FUNCTION_BLOCK "GCS7_E_MDDx_DP"	// FB 37
TITLE = MDDx Profibus Communication
//  
//COPYRIGHT:    (C) 1998  BUHLER AG, CH-9240 UZWIL, SWITZERLAND
//
//PRODUCT:      GCS7R1
//
//TITLE:        Element Control MDDx Profibus Communication
//
//REVISION:     11
//
//-------------------------------------------------------------------------
//
//IDENT:        AUTHOR:             DEPT:                      DATE:
//
//FB37.3.3      A. Egli             BASE                       30-Mar-2009
//              -PCD: OType=1037
//FB37.3.3      A. Egli             BASE                       16-Dec-2008
//              -Gap adjustement MDDR/T (GCS7R2 3.3)
//FB37.2.1      A. Egli             BASE                       25-Mar-2008
//              Len UDT SSW_MDDX_DP_Alarm is 6 Byte
//FB37.2.0      A. Egli             CT3                        25-Feb-2008
//              - New tagname for digital inputs Status.InpDI_0x
//              - Delete Status if OutComFault
//FB37.1.2      A. Egli             CT3                        21-Nov-2007
//              Message 42=A072CANDOUT
//FB37.1.1      A. Egli             CT3                        19-Nov-2006
//              Copy also AlarmNo > 74
//FB37.1.0      A. Egli             CT3                        11-Jun-2005
//              New Release R1
//
//-------------------------------------------------------------------------
//
//PURPOSE:      MANUAL : see [SSW-EL-MDDX_MAN_en]
//
//RESTRICTIONS: S7
//              ParFault and ParWarning may be set together!
//
//
//-------------------------------------------------------------------------
//=======================================================
//Log Message: 
//------------------------------------------------------
//
//=======================================================
//StCode:  State Communication               
//------------------------------------------------------
//43  StComFault.Local
// 3  StComOk                    
//32  StFault                 
//=======================================================
//StCode:  State Passage
//------------------------------------------------------
// 1  StDisengaged 
//11  StDisengaged.Warning 
//41  StDisengaged.DPFault
// 4  StEngaged
//14  StEngaged.Warning 
//44  StEngaged.DPFault
//32  StFault                 
//
//
AUTHOR : EA
FAMILY : GCS7LL
NAME : MDDxDP
VERSION : 3.4
VAR
  StCode : INT ;	//Element state code
  spare20 : BOOL ;
  spare21 : BOOL ;
  InOverrideHL : BOOL ;	//Override HL Inlet
  CmdNewJob : BOOL ;	//Send Target Value to LC, even if in manual mode
  CmdNewValue : BOOL ;	//Send Target Values
  spare25 : BOOL ;
  spare26 : BOOL ;
  spare27 : BOOL ;
  spare30 : BOOL ;
  spare31 : BOOL ;
  spare32 : BOOL ;
  CmdFaultReset : BOOL ;	//Command to reset fault
  InLocal : BOOL ;	//1= Local mode (no fault by start with service switch)
  spare35 : BOOL ;	//Warning is active
  spare36 : BOOL ;
  spare37 : BOOL ;
  InSimulation : BOOL ;	//Simulation with DPSim
  OutComFault : BOOL ;	//Communication fault
  VarEdgeStFault : BOOL ;
  OutWarning : BOOL ;
  OutFaultRelevant : BOOL ;	//Relavant faultfor group
  OutEdgeComFault : BOOL ;	//Alarm reason
  spare46 : BOOL ;
  spare47 : BOOL ;
  spare50 : BOOL ;
  spare51 : BOOL ;
  StOk : BOOL ;	//Element is ok
  spare53 : BOOL ;
  StFault : BOOL ;	//Element has a communication or device fault
  PCWrite : STRUCT
   Hsk : STRUCT
    AckRegisterSide1 : BOOL ;	//Acknowledge save recipe
    AckRollChangeDoneSide1 : BOOL ;	//Acknowledge roll change
    AckRegisterSide2 : BOOL ;	//Acknowledge save recipe
    AckRollChangeDoneSide2 : BOOL ;	//Acknowledge roll change
    Ack600CalibrationSide1 : BOOL ;	//Acknowledge 600 calibration
    Ack600CalibrationSide2 : BOOL ;	//Acknowledge 600 calibration
   END_STRUCT ;
  END_STRUCT ;
  PCRead : STRUCT
   Hsk : STRUCT
    ReqRegisterSide1 : BOOL ;	//Announcement save recipe
    ReqRollChangeDoneSide1 : BOOL ;	//Announcement roll change has be done
    ReqRegisterSide2 : BOOL ;	//Announcement save recipe
    ReqRollChangeDoneSide2 : BOOL ;	//Announcement roll change has be done
    Req600CalibrationSide1 : BOOL ;	//Announcement 600 calibration
    Req600CalibrationSide2 : BOOL ;	//Announcement 600 calibration
   END_STRUCT ;
  END_STRUCT ;
  Side1 : STRUCT
   StCode : INT ;
   InEnableDosing : BOOL ;	//Signal to engage the rolls and start dosing
   InRestdischarge : BOOL ;	//Signal to activate restdischarge mode
   CmdNewJob : BOOL ;	//Send Target Value to LC, even if in manual mode
   CmdNewValue : BOOL ;	//Send new Values to LC
   OutLCFault : BOOL ;	//LC has a relevant fault
   OutLCWarning : BOOL ;	//LC has a relevant fault
   OutAlarmNoValid : BOOL ;
   OutManual : BOOL ;	//LC Manual Mode
   VarEdgeStFault : BOOL ;
   StDisenaged : BOOL ;	//Element is ok
   StEngaged : BOOL ;	//Element is ok
   StFault : BOOL ;	//Element has a communication or device fault
   In : STRUCT 	//Only without MDEF
    InRollsUpCurrent : INT ;	//de: Aktuelle Stromaufnahme Motor 1 [0.1 A]
    InRollsLowCurrent : INT ;	//de: Aktuelle Stromaufnahme Motor 2 [0.1 A]
    InGapTopLeft : INT ;	//de:  Sollwert Mahlspalt oben links
    InGapTopRight : INT ;	//de:  Sollwert Mahlspalt oben rechts
    InGapBottomLeft : INT ;	//de:  Sollwert Mahlspalt unten links
    InGapBottomRight : INT ;	//de:  Sollwert Mahlspalt unten rechts
    InRollsLowUsed : BOOL ;	//MDDT: 1=Engage also lower rolls
    InRollsUpUsed : BOOL ;	//MDDT: 1=Engage also upper rolls
    InGapAdjustment : INT ;	//10=OFF,11=AUT,12=MAN,13=LOC,14=RCHG,0=nothing
   END_STRUCT ;
   Out : STRUCT 	//Only without MDEF
    OutRollsUpLoad : INT ;	//Is read from LC [%]
    OutRollsUpCurrent : INT ;	//Is read from LC [0.1 A]
    OutRollsLowLoad : INT ;	//Is read from LC [%]
    OutRollsLowCurrent : INT ;	//Is read from LC [0.1 A]
    OutFeedRollSpeed : INT ;	//Is read from LC [Hz]
    OutGrindingRollsUpSpeed : INT ;	//Is read from LC [0..999 RPM]
    OutGrindingRollsLowSpeed : INT ;	//Is read from LC [0..999 RPM]
    spare : INT ;
    OutAlarmNo : INT ;	//Is read from LC [0..9999]
    OutGapAdjustmentStatus : INT ;	//10=OFF,11=AUT,12=MAN,13=LOC,14=RCHG
    OutGapTopLeftAct : INT ;	//de:  Istwert Mahlspalt oben links
    OutGapTopRightAct : INT ;	//de:  Istwert Mahlspalt oben rechts
    OutGapBottomLeftAct : INT ;	//de:  Istwert Mahlspalt unten links
    OutGapBottomRightAct : INT ;	//de:  Istwert Mahlspalt unten rechts
    OutProductLevel : INT ;	//Is read from LC [+-500]
    OutTemperatureHoot : INT ;	//Is read from LC [°C]
    OutRunningTimeEngage : INT ;	//Is read from LC [h]
    OutRunningTimeRollsUp : INT ;	//Is read from LC [h]
    OutRunningTimeRollsLow : INT ;	//Is read from LC [h]
    OutCntEngage : INT ;	//Is read from LC []
    OutStatus : STRUCT 	//Is read from LC
     OutMDDR : BOOL ;
     OutHLBackupLeft : BOOL ;
     OutHLBackupRight : BOOL ;
    END_STRUCT ;
    OutLCAlarm : UDT 20373;
    tmpLCAlarm : UDT 20373;
   END_STRUCT ;
   OutTimeFaulted : DINT ;	//[s] Not errasable time "Faulted"
   OutCntFault : DINT ;	//Not errasable counter of faults
  END_STRUCT ;
  Side2 : STRUCT
   StCode : INT ;
   InEnableDosing : BOOL ;	//Signal to engage the rolls and start dosing
   InRestdischarge : BOOL ;	//Signal to activate restdischarge mode
   CmdNewJob : BOOL ;	//Send Target Value to LC, even if in manual mode
   CmdNewValue : BOOL ;	//Send new Values to LC
   OutLCFault : BOOL ;	//LC has a relevant fault
   OutLCWarning : BOOL ;	//LC has a relevant fault
   OutAlarmNoValid : BOOL ;
   OutManual : BOOL ;	//LC Manual Mode
   VarEdgeStFault : BOOL ;
   StDisenaged : BOOL ;	//Element is ok
   StEngaged : BOOL ;	//Element is ok
   StFault : BOOL ;	//Element has a communication or device fault
   In : STRUCT 	//Only without MDEF
    InRollsUpCurrent : INT ;	//de: Aktuelle Stromaufnahme Motor 1 [0.1 A]
    InRollsLowCurrent : INT ;	//de: Aktuelle Stromaufnahme Motor 2 [0.1 A]
    InGapTopLeft : INT ;	//de:  Sollwert Mahlspalt oben links
    InGapTopRight : INT ;	//de:  Sollwert Mahlspalt oben rechts
    InGapBottomLeft : INT ;	//de:  Sollwert Mahlspalt unten links
    InGapBottomRight : INT ;	//de:  Sollwert Mahlspalt unten rechts
    InRollsLowUsed : BOOL ;	//MDDT: 1=Engage also lower rolls
    InRollsUpUsed : BOOL ;	//MDDT: 1=Engage also upper rolls
    InGapAdjustment : INT ;	//10=OFF,11=AUT,12=MAN,13=LOC,14=RCHG,0=nothing
   END_STRUCT ;
   Out : STRUCT 	//Only without MDEF
    OutRollsUpLoad : INT ;	//Is read from LC [%]
    OutRollsUpCurrent : INT ;	//Is read from LC [0.1 A]
    OutRollsLowLoad : INT ;	//Is read from LC [%]
    OutRollsLowCurrent : INT ;	//Is read from LC [0.1 A]
    OutFeedRollSpeed : INT ;	//Is read from LC [HZ]
    OutGrindingRollsUpSpeed : INT ;	//Is read from LC [0..999 RPM]
    OutGrindingRollsLowSpeed : INT ;	//Is read from LC [0..999 RPM]
    spare : INT ;
    OutAlarmNo : INT ;	//Is read from LC [0..9999]
    OutGapAdjustmentStatus : INT ;	//0=Off;1=Manual;2=Automatic;3=Referencing;4=Aligment;5=Save
    OutGapTopLeftAct : INT ;	//de:  Istwert Mahlspalt oben links
    OutGapTopRightAct : INT ;	//de:  Istwert Mahlspalt oben rechts
    OutGapBottomLeftAct : INT ;	//de:  Istwert Mahlspalt unten links
    OutGapBottomRightAct : INT ;	//de:  Istwert Mahlspalt unten rechts
    OutProductLevel : INT ;	//Is read from LC [+-500]
    OutTemperatureHoot : INT ;	//Is read from LC [°C]
    OutRunningTimeEngage : INT ;	//Is read from LC [h]
    OutRunningTimeRollsUp : INT ;	//Is read from LC [h]
    OutRunningTimeRollsLow : INT ;	//Is read from LC [h]
    OutCntEngage : INT ;	//Is read from LC []
    OutStatus : STRUCT 	//Is read from LC
     OutMDDR : BOOL ;
     OutHLBackupLeft : BOOL ;
     OutHLBackupRight : BOOL ;
    END_STRUCT ;
    OutLCAlarm : UDT 20373;
    tmpLCAlarm : UDT 20373;
   END_STRUCT ;
   OutTimeFaulted : DINT ;	//[s] Not errasable time "Faulted"
   OutCntFault : DINT ;	//Not errasable counter of faults
  END_STRUCT ;
  Side1Divide : STRUCT
   StCode : INT ;
   OutLCFault : BOOL ;	//LC has a relevant fault
   OutLCWarning : BOOL ;	//LC has a relevant fault
   OutAlarmNoValid : BOOL ;
   VarEdgeStFault : BOOL ;
   StDisenaged : BOOL ;	//Element is ok
   StEngaged : BOOL ;	//Element is ok
   StFault : BOOL ;	//Element has a communication or device fault
   Out : STRUCT
    OutProductLevel : INT ;	//Is read from LC [+-500]
    OutFeedRollSpeed : INT ;	//Is read from LC [0..999 RPM]
    OutHLInlet : BOOL ;	//de:Einlaufsonde Left
    OutAlarmNo : INT ;	//Is read from LC [0..9999]
    OutLCAlarm : UDT 20373;
    tmpLCAlarm : UDT 20373;
   END_STRUCT ;
   OutTimeFaulted : DINT ;	//[s] Not errasable time "Faulted"
   OutCntFault : DINT ;	//Not errasable counter of faults
  END_STRUCT ;
  Side2Divide : STRUCT
   StCode : INT ;
   OutLCFault : BOOL ;	//LC has a relevant fault
   OutLCWarning : BOOL ;	//LC has a relevant fault
   OutAlarmNoValid : BOOL ;
   VarEdgeStFault : BOOL ;
   StDisenaged : BOOL ;	//Element is ok
   StEngaged : BOOL ;	//Element is ok
   StFault : BOOL ;	//Element has a communication or device fault
   Out : STRUCT
    OutProductLevel : INT ;	//Is read from LC [+-500]
    OutFeedRollSpeed : INT ;	//Is read from LC [0..999 RPM]
    OutHLInlet : BOOL ;	//de:Einlaufsonde Left
    OutAlarmNo : INT ;	//Is read from LC [0..9999]
    OutLCAlarm : UDT 20373;
    tmpLCAlarm : UDT 20373;
   END_STRUCT ;
   OutTimeFaulted : DINT ;	//[s] Not errasable time "Faulted"
   OutCntFault : DINT ;	//Not errasable counter of faults
  END_STRUCT ;
  OutAlarmNoLog : INT ;	//Last textnumber send to log
  OutTimeFaulted : DINT ;	//[s] Not errasable time "Faulted"
  OutCntFault : DINT ;	//Not errasable counter of faults
  Command : STRUCT
   S1Start : BOOL ;	//de: Start/Stop Links
   spare01 : BOOL ;
   S1RestDischarge : BOOL ;	//de: Restentleeren Links
   spare03 : BOOL ;
   spare04 : BOOL ;
   S1AckNewGapStatus : BOOL ;	//Acknowledge reading data
   spare06 : BOOL ;
   AcceptNewDataReady : BOOL ;	//de: Quittierung neue Werte Bereit
   S2Start : BOOL ;	//de: Start/Stop Rechts
   spare11 : BOOL ;
   S2RestDischarge : BOOL ;	//de: Restentleeren Rechts
   spare13 : BOOL ;
   spare14 : BOOL ;
   S2AckNewGapStatus : BOOL ;	//Acknowledge reading data
   spare16 : BOOL ;
   spare17 : BOOL ;	//de: Quittierung neue Werte Bereit
   spare20 : BYTE ;
   CommandReady : BOOL ;	//de: Steuersignale gültig
   spare31 : BOOL ;
   spare32 : BOOL ;
   spare33 : BOOL ;
   spare34 : BOOL ;
   ResetAlarm : BOOL ;	//de: Alarm löschen
   NewSendData : BOOL ;	//de: Aenderung Sendedaten
   AcceptNewRcvData : BOOL ;	//de: Quittierung Aenderung Empfangsdatensatz
  END_STRUCT ;
  Status : STRUCT
   S1Operation : BOOL ;	//de: Betrieb
   S1Disengaged : BOOL ;	//de: 1=Ausgerückt
   S1RestdischargeLocal : BOOL ;	//de: 1=Restentleeren Local
   S1DisengagedManual : BOOL ;	//Rolls manually disengaged: 1=Manually disengaged
   S1EnableMotors : BOOL ;	//de: Freigabe Mahlmotoren
   spare05 : BOOL ;
   spare06 : BOOL ;
   NewDataReady : BOOL ;	//de: Neue Werte Bereit
   S2Operation : BOOL ;	//de: Betrieb
   S2Disengaged : BOOL ;	//de: 1=Ausgerückt
   S2RestdischargeLocal : BOOL ;	//de: 1=Restentleeren Local
   S2DisengagedManual : BOOL ;	//Rolls manually disengaged: 1=Manually disengaged
   S2EnableMotors : BOOL ;	//de: Freigabe Mahlmotoren
   spare15 : BOOL ;
   spare16 : BOOL ;
   spare17 : BOOL ;	//de: Neue Werte Bereit
   InpDI_0_4 : BOOL ;	//DI 0.4: Default: Side 1 HL Inlet
   InpDI_0_5 : BOOL ;	//DI 0.5: Default: Side 1 HL Outlet 1
   InpDI_0_6 : BOOL ;	//DI 0.6: Default: Side 1 HL Outlet 2
   InpDI_0_7 : BOOL ;	//DI 0.7: Default: Side 1 HL Outlet 3
   InpDI_0_16 : BOOL ;	//DI 0.16: Default: Side 2 HL Inlet
   InpDI_0_17 : BOOL ;	//DI 0.17: Default: Side 2 HL Outlet 1
   InpDI_0_18 : BOOL ;	//DI 0.18: Default: Side 2 HL Outlet 2
   InpDI_0_19 : BOOL ;	//DI 0.19: Default: Side 2 HL Outlet 3
   InpDI_0_0 : BOOL ;	//DI0.0 Terminal X5:2
   InpDI_0_1 : BOOL ;	//DI0.1 Terminal X5:3
   InpDI_0_2 : BOOL ;	//DI0.2 Terminal X5:4
   RemoteControl : BOOL ;	//de: Sollwertvorgabe Remote
   WrongValue : BOOL ;	//de: Falscher Sollwert
   SumFault : BOOL ;	//de: Sammelalarm
   AcceptNewSendData : BOOL ;	//de: Quittierung Aenderung Sendedaten
   NewRcvData : BOOL ;	//de: Aenderung Empfangsdaten
  END_STRUCT ;
  Par : STRUCT
   ParObjectNo : INT ;	//Is used for communication with PC, e.g. for message
   ParMsgType : INT ;	//Is used for message (translation of state)
   ParHornCode : INT ;	//Is used by horn module
   ParLogOff : BOOL ;	//Report is off
   ParSide1Divided : BOOL ;	//Side 1 is divided
   ParSide2Divided : BOOL ;	//Side 2 is divided
   ParFilter : UDT 20373;	//Filter to alarm 1=Ignore alarm
   ParFilterWarning : UDT 20373;	//Filter to set alarm type (0=Fault;Suspend/1=Warning)
   ParIOByteNo : INT ;	//PROFIBUS: Address of first input and output byte
   HelpFlags : STRUCT
    CmdNewValueS1 : BOOL ;
    CmdNewValueS2 : BOOL ;
    CmdFaultReset : BOOL ;
    OutTestNewAlarm : BOOL ;	//Aux. signal to retry fault message
    OutComFaultRead : BOOL ;
    OutComFaultSend : BOOL ;
   END_STRUCT ;
   OutNoSndDataSet : BYTE ;	//de: Nummer Sendedatensatz
   OutIdxSndDataSet : BYTE ;	//de: Index Sendedatensatz
   OutNoRcvDataSet : BYTE ;	//de: Nummer Sendedatensatz
   OutIdxRcvDataSet : BYTE ;	//de: Index Sendedatensatz
   spare1 : DINT ;
  END_STRUCT ;
END_VAR
VAR_TEMP
  tmpAddrOffset : DWORD ;	//store the Instance Pointer
  tmpLOGvalue : WORD ;	//LOG value
  tmpCommand : INT ;
  tmpFault : BOOL ;
  tmpWarning : BOOL ;
  tmpLocal : BOOL ;
  tmpHornOn : BOOL ;
  tmpSendDone : BOOL ;	//Send Index is Equal receive Index
  tmpBit : BOOL ;
  tmpPxFault : BOOL ;
  tmpPxWarning : BOOL ;
  tmpPxAlarmNoValid : BOOL ;
  tmpAllAlarmNoValide : BOOL ;
  tmpAddrParFilter : DWORD ;	//Pointer to ParFilter
  tmpAddrParFilterWarning : DWORD ;	//Pointer to ParFilterWarning
  tmpIdx : INT ;
  tmpNewAlarm : UDT 20373;
  tmpOldAlarm : UDT 20373;
  tmpParFilterWarning : UDT 20373;
  tmpInt : INT ;
  tmpAddr : WORD ;
  tmpAddrIO : DINT ;
  tmpReturn : INT ;
  DPData : STRUCT
   StatusCommand : DWORD ;
   NoSndDataSet : BYTE ;	//de: Nummer Sendedatensatz
   IdxSndDataSet : BYTE ;	//de: Index Sendedatensatz
   NoRcvDataSet : BYTE ;	//de: Nummer Empfangsdatensatz
   IdxRcvDataSet : BYTE ;	//de: Index Empfangsdatensatz
   Data : STRUCT
    Byte8_9 : INT ;
    Byte10_11 : INT ;
    Byte12_13 : INT ;
    Byte14_15 : INT ;
    Byte16_17 : INT ;
    Byte18_19 : INT ;
    Byte20_21 : INT ;
    Byte22 : BYTE ;
    Byte23 : BYTE ;
   END_STRUCT ;
  END_STRUCT ;
  DPData16 : STRUCT
   StatusCommand : DWORD ;
   NoSndDataSet : BYTE ;	//de: Nummer Sendedatensatz
   IdxSndDataSet : BYTE ;	//de: Index Sendedatensatz
   NoRcvDataSet : BYTE ;	//de: Nummer Empfangsdatensatz
   IdxRcvDataSet : BYTE ;	//de: Index Empfangsdatensatz
   Data : ARRAY  [1 .. 4 ] OF DINT ;
  END_STRUCT ;
  DPData_Alarm120 : ARRAY  [0 .. 127 ] OF BOOL ;
  DPData_Alarm121 : ARRAY  [127 .. 255 ] OF BOOL ;
  tmpAddrOut_OutLCAlarm : DWORD ;
  tmpAddrOut_tmpLCAlarm : DWORD ;
END_VAR
BEGIN
NETWORK
TITLE =  Start Global
      TAR2;
      L     DW#16#FFFFFF;
      AD;
      T     #tmpAddrOffset;	//-->Addr Para
      L     P##Par;	//[3.1]
      +D;	//[3.1]
      L     P#8.0;
      +D;
      T     #tmpAddrParFilter;	//-->Pointer to Par.ParFilter
      L     P#6.0;
      +D;
      T     #tmpAddrParFilterWarning;	//-->Pointer to Par.ParFilterWarning
      SET;
      R     #tmpHornOn;
NETWORK
TITLE = PC Control
//=== Test Object number =====================
      L     "SYS_DirectCtrlDB".PC.ObjectNo;	//PCControl.ObjectNo
      L     #Par.ParObjectNo;	//Input ObjectNo
      <>I;
      JC    Ctrl;
//=== Test OType      ========================
      L     1037;	//Input object type
      L     "SYS_DirectCtrlDB".PC.ObjectType;	//PCControl.ObjectType
      <>I;
      JC    Ctrl;
//=== Test Handshake =========================
      A     "SYS_DirectCtrlDB".PC.Hsk.FExamine;	// Handshake.FExamine
      JC    pExa;
      A     "SYS_DirectCtrlDB".PC.Hsk.FDefineCmd;	// Handshake.FDefineCmd
      JC    pCmd;
      A     "SYS_DirectCtrlDB".PC.Hsk.FDefinePara;	// Handshake.FDefinePara
      JC    pPar;
      JU    pIni;
pIni: L     2;	//FcInit
      UC    "SYS_DirectCtrl";
      JU    Ctrl;
//Write parameter 
pPar: NOP   0;
//Write new commands from PC to Interface of group 
pCmd: A     "SYS_DirectCtrlDB".PC.Cmd1[11];	//CmdFaultReset
      S     #CmdFaultReset;
//------------------------------------------
pExa: NOP   0;
      TAR2;	// Address Dynamic datas
      T     "SYS_DirectCtrlDB".GC.InDynAddr;	// -->PCControl.GC.InDynAddr
      L     288;	// Length Dynamic datas
      T     "SYS_DirectCtrlDB".GC.InDynLen;	// -->PCControl.GC.InDynLen
      L     0;
      T     "SYS_DirectCtrlDB".GC.InParaAddr;	// -->PCControl.GC.InParaAddr
      T     "SYS_DirectCtrlDB".GC.InParaLen;	// -->PCControl.GC.InParaLen
      L     1;	// Code FcExamine
      UC    "SYS_DirectCtrl";
      L     11;	//Revision
      T     "SYS_DirectCtrlDB".GC.Revision;
Ctrl: NOP   0;
NETWORK
TITLE = (Profibus) Read data and store Data 
      L     #Par.ParIOByteNo;
      T     #tmpAddr;
      A     #InSimulation;
      JC    rSim;
      CALL  "SIEMENS_DPRD_DAT" (
           LADDR                    := #tmpAddr,
           RET_VAL                  := #tmpReturn,
           RECORD                   := #DPData);
      L     #tmpReturn;
      L     0;
      <>I;
      =     #Par.HelpFlags.OutComFaultRead;
      JC    rcv0;
      JU    rDP;
//read from Simulation
rSim: R     #Par.HelpFlags.OutComFaultRead;
      A     "GCS7_Gr_SimDPtoImage";
      L     P#I 0.0;
      JC    rDB1;
      OPN   "TEST_IOSimuliInput";
      L     P#DBX 0.0;
rDB1: L     #Par.ParIOByteNo;
      SLD   3;
      +D;
      T     #tmpAddrIO;
      LAR1  #tmpAddrIO;
      L     D [AR1,P#0.0];
      T     #DPData.StatusCommand;
      LAR1  #tmpAddrIO;
      L     D [AR1,P#4.0];
      LAR1  P##DPData;
      T     LD [AR1,P#4.0];
      LAR1  #tmpAddrIO;
      L     D [AR1,P#8.0];
      LAR1  P##DPData;
      T     LD [AR1,P#8.0];
      LAR1  #tmpAddrIO;
      L     D [AR1,P#12.0];
      LAR1  P##DPData;
      T     LD [AR1,P#12.0];
      LAR1  #tmpAddrIO;
      L     D [AR1,P#16.0];
      LAR1  P##DPData;
      T     D [AR1,P#16.0];
      LAR1  #tmpAddrIO;
      L     D [AR1,P#20.0];
      LAR1  P##DPData;
      T     D [AR1,P#20.0];
//===Test Send Data
rDP:  L     #DPData.NoSndDataSet;
      L     #Par.OutNoSndDataSet;
      ==I;
      A(;
      L     #DPData.IdxSndDataSet;
      L     #Par.OutIdxSndDataSet;
      ==I;
      );
      =     #tmpSendDone;
//==Copy Status===============
      L     #DPData.NoRcvDataSet;
      L     0;
      ==I;
      JC    R01A;
      CALL  "SIEMENS_BLKMOV" (
           SRCBLK                   := #DPData.StatusCommand,
           RET_VAL                  := #tmpReturn,
           DSTBLK                   := #Status);
      AN    #Status.NewRcvData;
      A     #InSimulation;
      JC    rcv0;
//===============================
//Answer Dataset 001
      L     #DPData.NoRcvDataSet;
      L     1;
      <>I;
      JC    r02;
//Answer Dataset 001 Index 1
      L     #DPData.IdxRcvDataSet;
      L     1;
      <>I;
      JC    r01B;
      L     #DPData.Data.Byte8_9;
      T     #Side1.Out.OutRollsUpLoad;
      L     #DPData.Data.Byte10_11;
      T     #Side1.Out.OutRollsUpCurrent;
      L     #DPData.Data.Byte12_13;
      T     #Side1.Out.OutRollsLowLoad;
      L     #DPData.Data.Byte14_15;
      T     #Side1.Out.OutRollsLowCurrent;
      L     #DPData.Data.Byte16_17;
      T     #Side1.Out.OutFeedRollSpeed;
      L     #DPData.Data.Byte18_19;
      T     #Side1.Out.OutGrindingRollsUpSpeed;
      L     #DPData.Data.Byte20_21;
      T     #Side1.Out.OutGrindingRollsLowSpeed;
      L     #DPData.Data.Byte23;
      T     #Side1.Out.OutAlarmNo;
      JU    R01B;
//Answer Dataset 001 Index 2
r01B: L     #DPData.IdxRcvDataSet;
      L     2;
      <>I;
      JC    r01C;
      L     #DPData.Data.Byte8_9;
      T     #Side2.Out.OutRollsUpLoad;
      L     #DPData.Data.Byte10_11;
      T     #Side2.Out.OutRollsUpCurrent;
      L     #DPData.Data.Byte12_13;
      T     #Side2.Out.OutRollsLowLoad;
      L     #DPData.Data.Byte14_15;
      T     #Side2.Out.OutRollsLowCurrent;
      L     #DPData.Data.Byte16_17;
      T     #Side2.Out.OutFeedRollSpeed;
      L     #DPData.Data.Byte18_19;
      T     #Side2.Out.OutGrindingRollsUpSpeed;
      L     #DPData.Data.Byte20_21;
      T     #Side2.Out.OutGrindingRollsLowSpeed;
      L     #DPData.Data.Byte23;
      T     #Side2.Out.OutAlarmNo;
      JU    R01C;
//Answer Dataset 001 Index 3
r01C: L     #DPData.IdxRcvDataSet;
      L     3;
      <>I;
      JC    r02;
//--Side1 Ext
      L     #DPData.Data.Byte8_9;
      T     #Side1Divide.Out.OutProductLevel;
      L     #DPData.Data.Byte10_11;
      T     #Side1Divide.Out.OutFeedRollSpeed;
      L     #DPData.Data.Byte12_13;
      T     #Side1Divide.Out.OutAlarmNo;
      L     #DPData.Data.Byte23;
      L     2#1;
      AW;
      L     0;
      <>I;
      =     #Side1Divide.Out.OutHLInlet;
//--Side2 Ext
      L     #DPData.Data.Byte16_17;
      T     #Side2Divide.Out.OutProductLevel;
      L     #DPData.Data.Byte18_19;
      T     #Side2Divide.Out.OutFeedRollSpeed;
      L     #DPData.Data.Byte20_21;
      T     #Side2Divide.Out.OutAlarmNo;
      L     #DPData.Data.Byte23;
      L     2#10000;
      AW;
      L     0;
      <>I;
      =     #Side2Divide.Out.OutHLInlet;
      JU    R02A;
//===============================
//Answer Dataset 002
r02:  L     #DPData.NoRcvDataSet;
      L     2;
      <>I;
      JC    r03;
//Answer Dataset 002 Index 1
      L     #DPData.IdxRcvDataSet;
      L     1;
      <>I;
      JC    r02B;	//[5.0]
      L     #DPData.Data.Byte8_9;
      T     #Side1.Out.OutProductLevel;
      L     #DPData.Data.Byte10_11;
      T     #Side1.Out.OutTemperatureHoot;
      L     #DPData.Data.Byte12_13;
      T     #Side1.Out.OutRunningTimeEngage;
      L     #DPData.Data.Byte14_15;
      T     #Side1.Out.OutRunningTimeRollsUp;
      L     #DPData.Data.Byte16_17;
      T     #Side1.Out.OutRunningTimeRollsLow;
      L     #DPData.Data.Byte18_19;
      T     #Side1.Out.OutCntEngage;
      CALL  "SIEMENS_BLKMOV" (
           SRCBLK                   := #DPData.Data.Byte20_21,
           RET_VAL                  := #tmpInt,
           DSTBLK                   := #Side1.Out.OutStatus);
      JU    R02B;
//Answer Dataset 002 Index 1
r02B: L     #DPData.IdxRcvDataSet;
      L     2;
      <>I;
      JC    r03;	//[5.0]
      L     #DPData.Data.Byte8_9;
      T     #Side2.Out.OutProductLevel;
      L     #DPData.Data.Byte10_11;
      T     #Side2.Out.OutTemperatureHoot;
      L     #DPData.Data.Byte12_13;
      T     #Side2.Out.OutRunningTimeEngage;
      L     #DPData.Data.Byte14_15;
      T     #Side2.Out.OutRunningTimeRollsUp;
      L     #DPData.Data.Byte16_17;
      T     #Side2.Out.OutRunningTimeRollsLow;
      L     #DPData.Data.Byte18_19;
      T     #Side2.Out.OutCntEngage;
      CALL  "SIEMENS_BLKMOV" (
           SRCBLK                   := #DPData.Data.Byte20_21,
           RET_VAL                  := #tmpInt,
           DSTBLK                   := #Side2.Out.OutStatus);
      JU    R03A;
//===============================
//Answer Dataset 003
r03:  L     #DPData.NoRcvDataSet;
      L     3;
      <>I;
      JC    r11;
//Answer Dataset 003 Index 1
      L     #DPData.IdxRcvDataSet;
      L     1;
      <>I;
      JC    r03B;	//[5.0]
      L     2#100000000;
      L     #DPData.Data.Byte8_9;
      AW;
      ==I;
      =     #PCRead.Hsk.ReqRegisterSide1;
      AN    #PCRead.Hsk.ReqRegisterSide1;
      R     #PCWrite.Hsk.AckRegisterSide1;
      L     2#1000000000;
      L     #DPData.Data.Byte8_9;
      AW;
      ==I;
      =     #PCRead.Hsk.ReqRollChangeDoneSide1;
      AN    #PCRead.Hsk.ReqRollChangeDoneSide1;
      R     #PCWrite.Hsk.AckRollChangeDoneSide1;
      L     2#10000000000;
      L     #DPData.Data.Byte8_9;
      AW;
      ==I;
      =     #PCRead.Hsk.Req600CalibrationSide1;
      AN    #PCRead.Hsk.Req600CalibrationSide1;
      R     #PCWrite.Hsk.Ack600CalibrationSide1;
      L     #DPData.Data.Byte10_11;
      SRW   8;
      T     #Side1.Out.OutGapAdjustmentStatus;
      L     #DPData.Data.Byte12_13;
      T     #Side1.Out.OutGapTopLeftAct;
      L     #DPData.Data.Byte14_15;
      T     #Side1.Out.OutGapTopRightAct;
      L     #DPData.Data.Byte16_17;
      T     #Side1.Out.OutGapBottomLeftAct;
      L     #DPData.Data.Byte18_19;
      T     #Side1.Out.OutGapBottomRightAct;
      JU    R03B;
//Answer Dataset 002 Index 1
r03B: L     #DPData.IdxRcvDataSet;
      L     2;
      <>I;
      JC    r11;	//[5.0]
      L     2#100000000;
      L     #DPData.Data.Byte8_9;
      AW;
      ==I;
      =     #PCRead.Hsk.ReqRegisterSide2;
      AN    #PCRead.Hsk.ReqRegisterSide2;
      R     #PCWrite.Hsk.AckRegisterSide2;
      L     2#1000000000;
      L     #DPData.Data.Byte8_9;
      AW;
      ==I;
      =     #PCRead.Hsk.ReqRollChangeDoneSide2;
      AN    #PCRead.Hsk.ReqRollChangeDoneSide2;
      R     #PCWrite.Hsk.AckRollChangeDoneSide2;
      L     2#10000000000;
      L     #DPData.Data.Byte8_9;
      AW;
      ==I;
      =     #PCRead.Hsk.Req600CalibrationSide2;
      AN    #PCRead.Hsk.Req600CalibrationSide2;
      R     #PCWrite.Hsk.Ack600CalibrationSide2;
      L     #DPData.Data.Byte10_11;
      SRW   8;
      T     #Side2.Out.OutGapAdjustmentStatus;
      L     #DPData.Data.Byte12_13;
      T     #Side2.Out.OutGapTopLeftAct;
      L     #DPData.Data.Byte14_15;
      T     #Side2.Out.OutGapTopRightAct;
      L     #DPData.Data.Byte16_17;
      T     #Side2.Out.OutGapBottomLeftAct;
      L     #DPData.Data.Byte18_19;
      T     #Side2.Out.OutGapBottomRightAct;
      JU    R11;
//===Answer  dataset 11 ====
//===Answer  dataset 12 ====
r11:  L     #DPData.NoRcvDataSet;
      L     11;
      <>I;
      JC    rLCB;
      CALL  "SIEMENS_BLKMOV" (
           SRCBLK                   := #DPData.Data,
           RET_VAL                  := #tmpReturn,
           DSTBLK                   := #DPData16.Data);
// Answer Dataset 11
      L     '  ';
      T     "SYS_DirectCtrlLCDB".PC.Value[1];
      L     #DPData16.Data[1];
      T     DB10.DBD 60;
      L     #DPData16.Data[2];
      T     DB10.DBD 64;
      L     #DPData16.Data[3];
      T     DB10.DBD 68;
      L     #DPData16.Data[4];
      T     DB10.DBD 72;
      L     #DPData.IdxRcvDataSet;
      L     255;
      ==I;
      JC    rLCE;
      S     "SYS_DirectCtrlLCDB".GC.Set11Done;
      L     12;
      T     #DPData.NoRcvDataSet;
      L     0;
      T     #DPData.IdxRcvDataSet;
      JU    rcv0;	//--> Read dataset 12
// Answer Dataset 12
rLCB: L     #DPData.NoRcvDataSet;
      L     12;
      <>I;
      JC    r120;
      CALL  "SIEMENS_BLKMOV" (
           SRCBLK                   := #DPData.Data,
           RET_VAL                  := #tmpReturn,
           DSTBLK                   := #DPData16.Data);
      L     #DPData16.Data[1];
      T     DB10.DBD 76;
      L     #DPData16.Data[2];
      T     DB10.DBD 80;
      L     #DPData16.Data[3];
      T     DB10.DBD 84;
      L     #DPData16.Data[4];
      T     DB10.DBD 86;
      AN    "SYS_DirectCtrlLCDB".GC.Set11Done;
      JC    R20A;
rLCE: L     12;
      CALL  "SYS_DirectCtrl";
      JU    R20A;
//===========================================================
//Answer Dataset 120
//===========================================================
r120: L     #DPData.NoRcvDataSet;
      L     120;
      <>I;
      JC    r121;
      CALL  "SIEMENS_BLKMOV" (
           SRCBLK                   := #DPData.Data,
           RET_VAL                  := #tmpReturn,
           DSTBLK                   := #DPData_Alarm120);
      L     #DPData.IdxRcvDataSet;
      L     2;
      ==I;
      JC    r20B;
//Anserw Dataset 120 Side 1
      A     #DPData_Alarm120[1];	//A001Eprom
      O     #DPData_Alarm120[2];	//A002RAM
      O     #DPData_Alarm120[3];	//A003RTIME
      O     #DPData_Alarm120[4];	//A004SWDog
      O     #DPData_Alarm120[6];	//A006LostMemory
      O     #DPData_Alarm120[79];	//A079Software
      =     #Side1.Out.OutLCAlarm.AxxxSoftware;
      A     #DPData_Alarm120[12];	//A012HOSTCOM
      O     #DPData_Alarm120[14];	//A014Profibus
      =     #Side1.Out.OutLCAlarm.AxxxCommunication;
      A     #DPData_Alarm120[13];	//A013EXPDISP
      O     #DPData_Alarm120[17];	//W017DISPLAY
      =     #Side1.Out.OutLCAlarm.AxxxDisplay;
      A     #DPData_Alarm120[5];
      =     #Side1.Out.OutLCAlarm.A005No24V;
      A     #DPData_Alarm120[7];
      =     #Side1.Out.OutLCAlarm.Ax07Range;
      A     #DPData_Alarm120[18];
      =     #Side1.Out.OutLCAlarm.A018Battery;
      A     #DPData_Alarm120[24];
      =     #Side1.Out.OutLCAlarm.A024Empty;
      A     #DPData_Alarm120[30];
      =     #Side1.Out.OutLCAlarm.Ax30Zero;
      A     #DPData_Alarm120[32];
      =     #Side1.Out.OutLCAlarm.Ax32ROD;
      A     #DPData_Alarm120[50];
      =     #Side1.Out.OutLCAlarm.Ax50FRoll1;
      A     #DPData_Alarm120[51];
      =     #Side1.Out.OutLCAlarm.Ax51FRoll2;
      A     #DPData_Alarm120[52];
      =     #Side1.Out.OutLCAlarm.A052RollUp;
      A     #DPData_Alarm120[53];
      =     #Side1.Out.OutLCAlarm.A053RollLow;
      A     #DPData_Alarm120[54];
      =     #Side1.Out.OutLCAlarm.A054MotUp;
      A     #DPData_Alarm120[55];
      =     #Side1.Out.OutLCAlarm.A055MotLow;
      A     #DPData_Alarm120[56];
      =     #Side1.Out.OutLCAlarm.A056STBYUP;
      A     #DPData_Alarm120[57];
      =     #Side1.Out.OutLCAlarm.A057STBYDN;
      A     #DPData_Alarm120[58];
      =     #Side1.Out.OutLCAlarm.A058M_Stop;
      A     #DPData_Alarm120[59];
      =     #Side1.Out.OutLCAlarm.A059M_Stop;
      A     #DPData_Alarm120[60];
      =     #Side1.Out.OutLCAlarm.Ax60HLInlet;
      A     #DPData_Alarm120[61];
      =     #Side1.Out.OutLCAlarm.A061HLOut1;
      A     #DPData_Alarm120[62];
      =     #Side1.Out.OutLCAlarm.A062HLOut2;
      A     #DPData_Alarm120[63];
      =     #Side1.Out.OutLCAlarm.A063HLOut3;
      A     #DPData_Alarm120[64];
      =     #Side1.Out.OutLCAlarm.A064HLBackupLeft;
      A     #DPData_Alarm120[65];
      =     #Side1.Out.OutLCAlarm.W065HLBackupLeft;
      A     #DPData_Alarm120[66];
      =     #Side1.Out.OutLCAlarm.A066HLBackupRight;
      A     #DPData_Alarm120[67];
      =     #Side1.Out.OutLCAlarm.W067HLBackupRight;
      A     #DPData_Alarm120[68];
      =     #Side1.Out.OutLCAlarm.Ax68InletFull;
      A     #DPData_Alarm120[69];
      =     #Side1.Out.OutLCAlarm.Ax69DosMax;
      A     #DPData_Alarm120[70];
      =     #Side1.Out.OutLCAlarm.A070CANCOM;
      A     #DPData_Alarm120[71];
      =     #Side1.Out.OutLCAlarm.A071CANMOD;
      A     #DPData_Alarm120[72];
      =     #Side1.Out.OutLCAlarm.A072CANDOUT;
      A     #DPData_Alarm120[75];
      =     #Side1.Out.OutLCAlarm.W075WarnTemp;
      A     #DPData_Alarm120[76];
      =     #Side1.Out.OutLCAlarm.A076HighTemp;
      A     #DPData_Alarm120[77];
      =     #Side1.Out.OutLCAlarm.A077DigOut;
      A     #DPData_Alarm120[78];
      =     #Side1.Out.OutLCAlarm.A078Service;
      A     #DPData_Alarm120[110];
      =     #Side1.Out.OutLCAlarm.A110Gap;
      A     #DPData_Alarm120[107];
      =     #Side1Divide.Out.OutLCAlarm.Ax07Range;
      SET;
      R     #DPData_Alarm120[1];	//A001Eprom
      R     #DPData_Alarm120[2];	//A002RAM
      R     #DPData_Alarm120[3];	//A003RTIME
      R     #DPData_Alarm120[4];	//A004SWDog
      R     #DPData_Alarm120[6];	//A006LostMemory
      R     #DPData_Alarm120[5];	//A005No24V
      R     #DPData_Alarm120[7];	//Ax07Range
      R     #DPData_Alarm120[12];	//A012HOSTCOM
      R     #DPData_Alarm120[13];	//A013EXPDISP
      R     #DPData_Alarm120[14];	//A014Profibus
      R     #DPData_Alarm120[17];	//W017DISPLAY
      R     #DPData_Alarm120[18];	//A018Battery
      R     #DPData_Alarm120[24];	//A024Empty
      R     #DPData_Alarm120[30];	//Ax30Zero
      R     #DPData_Alarm120[32];	//Ax32ROD
      R     #DPData_Alarm120[50];	//A050FRoll1
      R     #DPData_Alarm120[51];	//A051FRoll2
      R     #DPData_Alarm120[52];	//A052RollUp
      R     #DPData_Alarm120[53];	//A053RollLow
      R     #DPData_Alarm120[54];	//A054MotUp
      R     #DPData_Alarm120[55];	//A055MotLow
      R     #DPData_Alarm120[56];	//A056STBYUP
      R     #DPData_Alarm120[57];	//A057STBYDN
      R     #DPData_Alarm120[58];	//A058M_Stop
      R     #DPData_Alarm120[59];	//A059M_Stop
      R     #DPData_Alarm120[60];	//Ax60HLInlet
      R     #DPData_Alarm120[61];	//A061HLOut1
      R     #DPData_Alarm120[62];	//A062HLOut2
      R     #DPData_Alarm120[63];	//A063HLOut3
      R     #DPData_Alarm120[64];	//A064HLBackupLeft
      R     #DPData_Alarm120[65];	//W065HLBackupLeft
      R     #DPData_Alarm120[66];	//A066HLBackupRight
      R     #DPData_Alarm120[67];	//W067HLBackupRight
      R     #DPData_Alarm120[68];	//Ax68InletFull
      R     #DPData_Alarm120[69];	//Ax69DosMax
      R     #DPData_Alarm120[70];	//A070CANCOM
      R     #DPData_Alarm120[71];	//A071CANMOD
      R     #DPData_Alarm120[72];	//A072CANDOUT
      R     #DPData_Alarm120[75];	//W075WarnTemp
      R     #DPData_Alarm120[76];	//A076HighTemp
      R     #DPData_Alarm120[77];	//A077DigOut
      R     #DPData_Alarm120[78];	//A078Service
      R     #DPData_Alarm120[79];	//A079Software
      R     #DPData_Alarm120[110];	//A110Gap
      R     #DPData_Alarm120[107];	//Ax07Range
      LAR1  P##DPData_Alarm120;
      L     LD [AR1,P#0.0];
      L     LD [AR1,P#4.0];
      OD;
      L     LD [AR1,P#8.0];
      OD;
      L     LD [AR1,P#12.0];
      OD;
      L     0;
      <>D;
      =     #Side1.Out.OutLCAlarm.AxxxUnknown;
      SET;
      S     #Side1.OutAlarmNoValid;
      JU    R21A;	//-->Read Dataset 121 Index 1
//Answer Dataset 120 Side 2
r20B: A     #DPData_Alarm120[1];	//A001Eprom
      O     #DPData_Alarm120[2];	//A002RAM
      O     #DPData_Alarm120[3];	//A003RTIME
      O     #DPData_Alarm120[4];	//A004SWDog
      O     #DPData_Alarm120[6];	//A006LostMemory
      O     #DPData_Alarm120[79];	//A079Software
      =     #Side2.Out.OutLCAlarm.AxxxSoftware;
      A     #DPData_Alarm120[12];	//A012HOSTCOM
      O     #DPData_Alarm120[14];	//A014Profibus
      =     #Side2.Out.OutLCAlarm.AxxxCommunication;
      A     #DPData_Alarm120[13];	//A013EXPDISP
      O     #DPData_Alarm120[17];	//W017DISPLAY
      =     #Side2.Out.OutLCAlarm.AxxxDisplay;
      A     #DPData_Alarm120[5];
      =     #Side2.Out.OutLCAlarm.A005No24V;
      A     #DPData_Alarm120[7];
      =     #Side2.Out.OutLCAlarm.Ax07Range;
      A     #DPData_Alarm120[18];
      =     #Side2.Out.OutLCAlarm.A018Battery;
      A     #DPData_Alarm120[24];
      =     #Side2.Out.OutLCAlarm.A024Empty;
      A     #DPData_Alarm120[30];
      =     #Side2.Out.OutLCAlarm.Ax30Zero;
      A     #DPData_Alarm120[32];
      =     #Side2.Out.OutLCAlarm.Ax32ROD;
      A     #DPData_Alarm120[50];
      =     #Side2.Out.OutLCAlarm.Ax50FRoll1;
      A     #DPData_Alarm120[51];
      =     #Side2.Out.OutLCAlarm.Ax51FRoll2;
      A     #DPData_Alarm120[52];
      =     #Side2.Out.OutLCAlarm.A052RollUp;
      A     #DPData_Alarm120[53];
      =     #Side2.Out.OutLCAlarm.A053RollLow;
      A     #DPData_Alarm120[54];
      =     #Side2.Out.OutLCAlarm.A054MotUp;
      A     #DPData_Alarm120[55];
      =     #Side2.Out.OutLCAlarm.A055MotLow;
      A     #DPData_Alarm120[56];
      =     #Side2.Out.OutLCAlarm.A056STBYUP;
      A     #DPData_Alarm120[57];
      =     #Side2.Out.OutLCAlarm.A057STBYDN;
      A     #DPData_Alarm120[58];
      =     #Side2.Out.OutLCAlarm.A058M_Stop;
      A     #DPData_Alarm120[59];
      =     #Side2.Out.OutLCAlarm.A059M_Stop;
      A     #DPData_Alarm120[60];
      =     #Side2.Out.OutLCAlarm.Ax60HLInlet;
      A     #DPData_Alarm120[61];
      =     #Side2.Out.OutLCAlarm.A061HLOut1;
      A     #DPData_Alarm120[62];
      =     #Side2.Out.OutLCAlarm.A062HLOut2;
      A     #DPData_Alarm120[63];
      =     #Side2.Out.OutLCAlarm.A063HLOut3;
      A     #DPData_Alarm120[64];
      =     #Side2.Out.OutLCAlarm.A064HLBackupLeft;
      A     #DPData_Alarm120[65];
      =     #Side2.Out.OutLCAlarm.W065HLBackupLeft;
      A     #DPData_Alarm120[66];
      =     #Side2.Out.OutLCAlarm.A066HLBackupRight;
      A     #DPData_Alarm120[67];
      =     #Side2.Out.OutLCAlarm.W067HLBackupRight;
      A     #DPData_Alarm120[68];
      =     #Side2.Out.OutLCAlarm.Ax68InletFull;
      A     #DPData_Alarm120[69];
      =     #Side2.Out.OutLCAlarm.Ax69DosMax;
      A     #DPData_Alarm120[70];
      =     #Side2.Out.OutLCAlarm.A070CANCOM;
      A     #DPData_Alarm120[71];
      =     #Side2.Out.OutLCAlarm.A071CANMOD;
      A     #DPData_Alarm120[72];
      =     #Side2.Out.OutLCAlarm.A072CANDOUT;
      A     #DPData_Alarm120[75];
      =     #Side2.Out.OutLCAlarm.W075WarnTemp;
      A     #DPData_Alarm120[76];
      =     #Side2.Out.OutLCAlarm.A076HighTemp;
      A     #DPData_Alarm120[77];
      =     #Side2.Out.OutLCAlarm.A077DigOut;
      A     #DPData_Alarm120[78];
      =     #Side2.Out.OutLCAlarm.A078Service;
      A     #DPData_Alarm120[110];
      =     #Side2.Out.OutLCAlarm.A110Gap;
      A     #DPData_Alarm120[107];
      =     #Side2Divide.Out.OutLCAlarm.Ax07Range;
      SET;
      R     #DPData_Alarm120[1];	//A001Eprom
      R     #DPData_Alarm120[2];	//A002RAM
      R     #DPData_Alarm120[3];	//A003RTIME
      R     #DPData_Alarm120[4];	//A004SWDog
      R     #DPData_Alarm120[6];	//A006LostMemory
      R     #DPData_Alarm120[5];	//A005No24V
      R     #DPData_Alarm120[7];	//Ax07Range
      R     #DPData_Alarm120[12];	//A012HOSTCOM
      R     #DPData_Alarm120[13];	//A013EXPDISP
      R     #DPData_Alarm120[14];	//A014Profibus
      R     #DPData_Alarm120[17];	//W017DISPLAY
      R     #DPData_Alarm120[18];	//A018Battery
      R     #DPData_Alarm120[24];	//A024Empty
      R     #DPData_Alarm120[30];	//Ax30Zero
      R     #DPData_Alarm120[32];	//Ax32ROD
      R     #DPData_Alarm120[50];	//A050FRoll1
      R     #DPData_Alarm120[51];	//A051FRoll2
      R     #DPData_Alarm120[52];	//A052RollUp
      R     #DPData_Alarm120[53];	//A053RollLow
      R     #DPData_Alarm120[54];	//A054MotUp
      R     #DPData_Alarm120[55];	//A055MotLow
      R     #DPData_Alarm120[56];	//A056STBYUP
      R     #DPData_Alarm120[57];	//A057STBYDN
      R     #DPData_Alarm120[58];	//A058M_Stop
      R     #DPData_Alarm120[59];	//A059M_Stop
      R     #DPData_Alarm120[60];	//Ax60HLInlet
      R     #DPData_Alarm120[61];	//A061HLOut1
      R     #DPData_Alarm120[62];	//A062HLOut2
      R     #DPData_Alarm120[63];	//A063HLOut3
      R     #DPData_Alarm120[64];	//A064HLBackupLeft
      R     #DPData_Alarm120[65];	//W065HLBackupLeft
      R     #DPData_Alarm120[66];	//A066HLBackupRight
      R     #DPData_Alarm120[67];	//W067HLBackupRight
      R     #DPData_Alarm120[68];	//Ax68InletFull
      R     #DPData_Alarm120[69];	//Ax69DosMax
      R     #DPData_Alarm120[70];	//A070CANCOM
      R     #DPData_Alarm120[71];	//A071CANMOD
      R     #DPData_Alarm120[72];	//A072CANDOUT
      R     #DPData_Alarm120[75];	//W075WarnTemp
      R     #DPData_Alarm120[76];	//A076HighTemp
      R     #DPData_Alarm120[77];	//A077DigOut
      R     #DPData_Alarm120[78];	//A078Service
      R     #DPData_Alarm120[79];	//A079Software
      R     #DPData_Alarm120[110];	//A110Gap
      R     #DPData_Alarm120[107];	//Ax07Range
      LAR1  P##DPData_Alarm120;
      L     LD [AR1,P#0.0];
      L     LD [AR1,P#4.0];
      OD;
      L     LD [AR1,P#8.0];
      OD;
      L     LD [AR1,P#12.0];
      OD;
      L     0;
      <>D;
      =     #Side2.Out.OutLCAlarm.AxxxUnknown;
      SET;
      S     #Side2.OutAlarmNoValid;
      JU    R21B;	//-->Read Dataset 121 Index 2
//===================================
//Answer  dataset 121
//===================================
r121: L     #DPData.NoRcvDataSet;
      L     121;
      <>I;
      JC    r28A;
      CALL  "SIEMENS_BLKMOV" (
           SRCBLK                   := #DPData.Data,
           RET_VAL                  := #tmpReturn,
           DSTBLK                   := #DPData_Alarm121);
      L     #DPData.IdxRcvDataSet;
      L     2;
      ==I;
      JC    r21B;
//Anserw Dataset 120 Side 1
      A     #DPData_Alarm121[130];
      =     #Side1Divide.Out.OutLCAlarm.Ax30Zero;
      A     #DPData_Alarm121[132];
      =     #Side1Divide.Out.OutLCAlarm.Ax32ROD;
      A     #DPData_Alarm121[150];
      =     #Side1Divide.Out.OutLCAlarm.Ax50FRoll1;
      A     #DPData_Alarm121[151];
      =     #Side1Divide.Out.OutLCAlarm.Ax51FRoll2;
      A     #DPData_Alarm121[160];
      =     #Side1Divide.Out.OutLCAlarm.Ax60HLInlet;
      A     #DPData_Alarm121[168];
      =     #Side1Divide.Out.OutLCAlarm.Ax68InletFull;
      A     #DPData_Alarm121[169];
      =     #Side1Divide.Out.OutLCAlarm.Ax69DosMax;
      SET;
      R     #DPData_Alarm121[130];	//Ax30Zero
      R     #DPData_Alarm121[132];	//Ax32ROD
      R     #DPData_Alarm121[150];	//A050FRoll1
      R     #DPData_Alarm121[151];	//A051FRoll2
      R     #DPData_Alarm121[160];	//Ax60HLInlet
      R     #DPData_Alarm121[168];	//Ax68InletFull
      R     #DPData_Alarm121[169];	//Ax69DosMax
      LAR1  P##DPData_Alarm121;
      L     LD [AR1,P#0.0];
      L     LD [AR1,P#4.0];
      OD;
      L     LD [AR1,P#8.0];
      OD;
      L     LD [AR1,P#12.0];
      OD;
      L     0;
      <>D;
      =     #Side1Divide.Out.OutLCAlarm.AxxxUnknown;
      SET;
      S     #Side1Divide.OutAlarmNoValid;
      JU    R20B;	//[3.3] //-->Read Dataset 120 Index 2
//Anserw Dataset 121 Side 2
r21B: A     #DPData_Alarm121[130];
      =     #Side2Divide.Out.OutLCAlarm.Ax30Zero;
      A     #DPData_Alarm121[132];
      =     #Side2Divide.Out.OutLCAlarm.Ax32ROD;
      A     #DPData_Alarm121[150];
      =     #Side2Divide.Out.OutLCAlarm.Ax50FRoll1;
      A     #DPData_Alarm121[151];
      =     #Side2Divide.Out.OutLCAlarm.Ax51FRoll2;
      A     #DPData_Alarm121[160];
      =     #Side2Divide.Out.OutLCAlarm.Ax60HLInlet;
      A     #DPData_Alarm121[168];
      =     #Side2Divide.Out.OutLCAlarm.Ax68InletFull;
      A     #DPData_Alarm121[169];
      =     #Side2Divide.Out.OutLCAlarm.Ax69DosMax;
      SET;
      R     #DPData_Alarm121[130];	//Ax30Zero
      R     #DPData_Alarm121[132];	//Ax32ROD
      R     #DPData_Alarm121[150];	//A050FRoll1
      R     #DPData_Alarm121[151];	//A051FRoll2
      R     #DPData_Alarm121[160];	//Ax60HLInlet
      R     #DPData_Alarm121[168];	//Ax68InletFull
      R     #DPData_Alarm121[169];	//Ax69DosMax
      LAR1  P##DPData_Alarm121;
      L     LD [AR1,P#0.0];
      L     LD [AR1,P#4.0];
      OD;
      L     LD [AR1,P#8.0];
      OD;
      L     LD [AR1,P#12.0];
      OD;
      L     0;
      <>D;
      =     #Side2Divide.Out.OutLCAlarm.AxxxUnknown;
      SET;
      S     #Side2Divide.OutAlarmNoValid;
      JU    R28A;	//-->Read Dataset 128 Index 1
//===============================
//Answer  dataset 128
r28A: L     #DPData.NoRcvDataSet;
      L     128;
      <>I;
      JC    R01A;
      L     #DPData.IdxRcvDataSet;
      L     1;
      <>I;
      JC    r28B;
      JU    R28B;
r28B: L     #DPData.IdxRcvDataSet;
      L     2;
      <>I;
      JC    R01A;
      JU    R01A;
//===============================
//Read Dataset 001 Index 1
R01A: L     1;
      T     #DPData.NoRcvDataSet;
      L     1;
      T     #DPData.IdxRcvDataSet;
      JU    rcv0;
//===============================
//Read Dataset 001   Index 2
R01B: L     1;
      T     #DPData.NoRcvDataSet;
      L     2;
      T     #DPData.IdxRcvDataSet;
      JU    rcv0;
//===============================
//Read Dataset 001   Index 3
R01C: AN    #Par.ParSide1Divided;
      AN    #Par.ParSide2Divided;
      JC    R02A;
      L     1;
      T     #DPData.NoRcvDataSet;
      L     3;
      T     #DPData.IdxRcvDataSet;
      JU    rcv0;
//===============================
//Read Dataset 002 Index 1
R02A: L     2;
      T     #DPData.NoRcvDataSet;
      L     1;
      T     #DPData.IdxRcvDataSet;
      JU    rcv0;
//===============================
//Read Dataset 001   Index 2
R02B: L     2;
      T     #DPData.NoRcvDataSet;
      L     2;
      T     #DPData.IdxRcvDataSet;
      JU    rcv0;
//===============================
//Read Dataset 003 Index 1
R03A: L     3;
      T     #DPData.NoRcvDataSet;
      L     1;
      T     #DPData.IdxRcvDataSet;
      JU    rcv0;
//===============================
//Read Dataset 003   Index 2
R03B: L     3;
      T     #DPData.NoRcvDataSet;
      L     2;
      T     #DPData.IdxRcvDataSet;
      JU    rcv0;
//===============================
//LC Parameter: Reading dataset 11
R11:  L     "SYS_DirectCtrlLCDB".PC.ObjectNo;
      L     #Par.ParObjectNo;
      <>D;
      JC    R20A;
      AN    "SYS_DirectCtrlLCDB".PC.Hsk.FExamineFirst;
      AN    "SYS_DirectCtrlLCDB".PC.Hsk.FExamineNext;
      JC    R20A;
// -- Start Reading with Dataset 11
      L     11;
      T     #DPData.NoRcvDataSet;
      L     253;	//First
      A     "SYS_DirectCtrlLCDB".PC.Hsk.FExamineFirst;
      JC    rLC9;
      L     254;	//Next
rLC9: T     #DPData.IdxRcvDataSet;
      JU    rcv0;
//===============================
//Read Dataset 120   Index 1
R20A: L     120;
      T     #DPData.NoRcvDataSet;
      L     1;
      T     #DPData.IdxRcvDataSet;
      JU    rcv0;
//Read Dataset 121   Index 1
R21A: AN    #Par.ParSide1Divided;
      JC    R20B;
      L     121;
      T     #DPData.NoRcvDataSet;
      L     1;
      T     #DPData.IdxRcvDataSet;
      JU    rcv0;
//Read Dataset 120   Index 2
R20B: L     120;
      T     #DPData.NoRcvDataSet;
      L     2;
      T     #DPData.IdxRcvDataSet;
      JU    rcv0;
//Read Dataset 121   Index 2
R21B: AN    #Par.ParSide2Divided;
      JC    R28A;
      L     121;
      T     #DPData.NoRcvDataSet;
      L     2;
      T     #DPData.IdxRcvDataSet;
      JU    rcv0;
//===============================
//Read Dataset 128 Index 1
R28A: JU    R01A;
      L     128;
      T     #DPData.NoRcvDataSet;
      L     1;
      T     #DPData.IdxRcvDataSet;
      JU    rcv0;
R28B: L     128;
      T     #DPData.NoRcvDataSet;
      L     2;
      T     #DPData.IdxRcvDataSet;
      JU    rcv0;
//===============================
rcv0: NOP   0;
NETWORK
TITLE =  All State Init
//===Clear tmp Variable
//===Global Group Orders===
      A     #InLocal;
      =     #tmpLocal;
//---Force Off------
//---FaultReset is on---
      A     "GCS7_Gr_OutFaultReset";	//Gr.OutFaultReset
      S     #CmdFaultReset;
//---CmdNewJob
      A     #CmdNewJob;
      S     #Side1.CmdNewJob;
      S     #Side2.CmdNewJob;
      R     #CmdNewJob;
//---CmdNewValue
      A     #CmdNewValue;
      S     #Side1.CmdNewValue;
      S     #Side2.CmdNewValue;
      R     #CmdNewValue;
//OutManual
      L     #Side1.Out.OutGapAdjustmentStatus;
      L     12;	//Manual
      ==I;
      =     #Side1.OutManual;
      L     #Side2.Out.OutGapAdjustmentStatus;
      L     12;	//Manual
      ==I;
      =     #Side2.OutManual;
//OutComFault
      A     #Par.HelpFlags.OutComFaultRead;
      O     #Par.HelpFlags.OutComFaultSend;
      =     #OutComFault;
//Init Signal IF ComFault      [2.0]
      AN    #OutComFault;	//[2.0]
      JC    ALJ0;	//[2.0]
      L     0;	//[2.0]
      T     #tmpInt;	//[2.0]
      CALL  "SIEMENS_FILL" (
           BVAL                     := #tmpInt,
           RET_VAL                  := #tmpIdx,
           BLK                      := #Status);	//[2.0]
ALJ0: NOP   0;
NETWORK
TITLE = Analyse Alarm and Log Entry
      L     1;
LAJ0: T     #tmpIdx;
      L     1;
      <>I;
      JC    LAP2;
      CALL  "SYS_BitAddress" (
           Source                   := #Side1.Out.OutLCAlarm,
           OutBitAddr               := #tmpAddrOut_OutLCAlarm);
      A     #Side1.OutAlarmNoValid;
      =     #tmpPxAlarmNoValid;
      JU    LAJ1;
LAP2: L     2;	//Passage Right
      L     #tmpIdx;
      <>I;
      JC    LAP3;
      CALL  "SYS_BitAddress" (
           Source                   := #Side2.Out.OutLCAlarm,
           OutBitAddr               := #tmpAddrOut_OutLCAlarm);
      A     #Side2.OutAlarmNoValid;
      =     #tmpPxAlarmNoValid;
      JU    LAJ1;
LAP3: L     3;	//Passage Divide Left
      L     #tmpIdx;
      <>I;
      JC    LAP4;
      CALL  "SYS_BitAddress" (
           Source                   := #Side1Divide.Out.OutLCAlarm,
           OutBitAddr               := #tmpAddrOut_OutLCAlarm);
      A     #Side1Divide.OutAlarmNoValid;
      =     #tmpPxAlarmNoValid;
      JU    LAJ1;
LAP4: L     4;	//Passage Divide Right
      L     #tmpIdx;
      <>I;
      JC    LAJ9;
      CALL  "SYS_BitAddress" (
           Source                   := #Side2Divide.Out.OutLCAlarm,
           OutBitAddr               := #tmpAddrOut_OutLCAlarm);
      A     #Side2Divide.OutAlarmNoValid;
      =     #tmpPxAlarmNoValid;
      JU    LAJ1;
//Check Alarm Mumber
LAJ1: NOP   0;
//--------------------------------------------
//Copy New Alarm from current index to stack tmpNewAlarm
      L     #tmpAddrOut_OutLCAlarm;
      L     P#6.0;	//[2.1]
      +D;
      T     #tmpAddrOut_tmpLCAlarm;
      LAR1  #tmpAddrOut_OutLCAlarm;
      L     DID [AR1,P#0.0];
      LAR1  #tmpAddrParFilter;
      L     DID [AR1,P#0.0];	//#Par.ParFilter;
      INVD;	//Invers filter mask
      AD;	//Resetfiltered bits
      LAR1  P##tmpNewAlarm;
      T     LD [AR1,P#0.0];	//-->tmpNewAlarm 
      LAR1  #tmpAddrOut_OutLCAlarm;
      L     DIW [AR1,P#4.0];
      LAR1  #tmpAddrParFilter;
      L     DIW [AR1,P#4.0];	//#Par.ParFilter;
      INVD;	//Invers filter mask
      AD;	//Resetfiltered bits
      LAR1  P##tmpNewAlarm;
      T     LW [AR1,P#4.0];	//-->tmpNewAlarm 
//Copy Old Alarm from current index to stack tmpOldAlarm
      LAR1  #tmpAddrOut_tmpLCAlarm;
      L     DID [AR1,P#0.0];
      LAR1  P##tmpOldAlarm;
      T     LD [AR1,P#0.0];	//tmpOldAlarm 
      LAR1  #tmpAddrOut_tmpLCAlarm;
      L     DIW [AR1,P#4.0];
      LAR1  P##tmpOldAlarm;
      T     LW [AR1,P#4.0];	//tmpOldAlarm 
//Copy Par.ParFilterWarning to tmpParFilterWarning;
      LAR1  #tmpAddrParFilterWarning;
      L     DID [AR1,P#0.0];	//Par.ParFilterWarning
      LAR1  P##tmpParFilterWarning;
      T     LD [AR1,P#0.0];	//tmpParFilterWarning
      LAR1  #tmpAddrParFilterWarning;
      L     DIW [AR1,P#4.0];	//Par.ParFilterWarning
      LAR1  P##tmpParFilterWarning;
      T     LW [AR1,P#4.0];	//tmpParFilterWarning
      A     #InOverrideHL;
      S     #tmpParFilterWarning.Ax60HLInlet;
//-------------
      LAR1  P##tmpNewAlarm;
      L     LD [AR1,P#0.0];	//-->tmpNewAlarm 
      LAR1  P##tmpParFilterWarning;
      L     LD [AR1,P#0.0];	//tmpParFilterWarning
      INVD;	//Invers filter mask
      AD;
      L     0;
      <>D;
      O(;
      LAR1  P##tmpNewAlarm;
      L     LW [AR1,P#4.0];	//-->tmpNewAlarm 
      LAR1  P##tmpParFilterWarning;
      L     LW [AR1,P#4.0];	//tmpParFilterWarning
      INVD;	//Invers filter mask
      AD;
      L     0;
      <>D;
      );
      =     #tmpPxFault;
      LAR1  P##tmpNewAlarm;
      L     LD [AR1,P#0.0];	//-->tmpNewAlarm 
      LAR1  P##tmpParFilterWarning;
      L     LD [AR1,P#0.0];	//tmpParFilterWarning
      AD;
      L     0;
      <>D;
      O(;
      LAR1  P##tmpNewAlarm;
      L     LW [AR1,P#0.0];	//-->tmpNewAlarm 
      LAR1  P##tmpParFilterWarning;
      L     LW [AR1,P#0.0];	//#Par.ParFilterWarning;
      AD;
      L     0;
      <>D;
      );
      =     #tmpPxWarning;
//-------------
//Check New Message
      A     #tmpPxFault;
      A     #tmpPxAlarmNoValid;
      AN    #tmpLocal;
      JC    LANM;
//Clear old Message
      L     0;
      LAR1  P##tmpOldAlarm;
      T     LD [AR1,P#0.0];
      JU    LAST;	//-Store Data
//-------------
LANM: L     B#(4, 1);
      A     #tmpNewAlarm.AxxxSoftware;
      FP    #tmpOldAlarm.AxxxSoftware;
      JC    LALG;
      L     B#(4, 2);
      A     #tmpNewAlarm.AxxxCommunication;
      FP    #tmpOldAlarm.AxxxCommunication;
      JC    LALG;
      L     B#(4, 3);
      A     #tmpNewAlarm.AxxxDisplay;
      FP    #tmpOldAlarm.AxxxDisplay;
      JC    LALG;
      L     B#(4, 4);
      A     #tmpNewAlarm.AxxxUnknown;
      FP    #tmpOldAlarm.AxxxUnknown;
      JC    LALG;
      L     B#(4, 5);
      A     #tmpNewAlarm.A005No24V;
      FP    #tmpOldAlarm.A005No24V;
      JC    LALG;
      L     B#(4, 7);
      A     #tmpNewAlarm.Ax07Range;
      FP    #tmpOldAlarm.Ax07Range;
      JC    LALG;
      L     B#(4, 18);
      A     #tmpNewAlarm.A018Battery;
      FP    #tmpOldAlarm.A018Battery;
      JC    LALG;
      L     B#(4, 9);
      A     #tmpNewAlarm.A024Empty;
      FP    #tmpOldAlarm.A024Empty;
      JC    LALG;
      L     B#(4, 10);
      A     #tmpNewAlarm.Ax30Zero;
      FP    #tmpOldAlarm.Ax30Zero;
      JC    LALG;
      L     B#(4, 12);
      A     #tmpNewAlarm.Ax32ROD;
      FP    #tmpOldAlarm.Ax32ROD;
      JC    LALG;
      L     B#(4, 20);
      A     #tmpNewAlarm.Ax50FRoll1;
      FP    #tmpOldAlarm.Ax50FRoll1;
      JC    LALG;
      L     B#(4, 21);
      A     #tmpNewAlarm.Ax51FRoll2;
      FP    #tmpOldAlarm.Ax51FRoll2;
      JC    LALG;
      L     B#(4, 22);
      A     #tmpNewAlarm.A052RollUp;
      FP    #tmpOldAlarm.A052RollUp;
      JC    LALG;
      L     B#(4, 23);
      A     #tmpNewAlarm.A053RollLow;
      FP    #tmpOldAlarm.A053RollLow;
      JC    LALG;
      L     B#(4, 24);
      A     #tmpNewAlarm.A054MotUp;
      FP    #tmpOldAlarm.A054MotUp;
      JC    LALG;
      L     B#(4, 25);
      A     #tmpNewAlarm.A055MotLow;
      FP    #tmpOldAlarm.A055MotLow;
      JC    LALG;
      L     B#(4, 26);
      A     #tmpNewAlarm.A056STBYUP;
      FP    #tmpOldAlarm.A056STBYUP;
      JC    LALG;
      L     B#(4, 27);
      A     #tmpNewAlarm.A057STBYDN;
      FP    #tmpOldAlarm.A057STBYDN;
      JC    LALG;
      L     B#(4, 28);
      A     #tmpNewAlarm.A058M_Stop;
      FP    #tmpOldAlarm.A058M_Stop;
      JC    LALG;
      L     B#(4, 29);
      A     #tmpNewAlarm.A059M_Stop;
      FP    #tmpOldAlarm.A059M_Stop;
      JC    LALG;
      L     B#(4, 30);
      A     #tmpNewAlarm.Ax60HLInlet;
      FP    #tmpOldAlarm.Ax60HLInlet;
      JC    LALG;
      L     B#(4, 31);
      A     #tmpNewAlarm.A061HLOut1;
      FP    #tmpOldAlarm.A061HLOut1;
      JC    LALG;
      L     B#(4, 32);
      A     #tmpNewAlarm.A062HLOut2;
      FP    #tmpOldAlarm.A062HLOut2;
      JC    LALG;
      L     B#(4, 33);
      A     #tmpNewAlarm.A063HLOut3;
      FP    #tmpOldAlarm.A063HLOut3;
      JC    LALG;
      L     B#(4, 34);
      A     #tmpNewAlarm.A064HLBackupLeft;
      FP    #tmpOldAlarm.A064HLBackupLeft;
      JC    LALG;
      L     B#(4, 35);
      A     #tmpNewAlarm.W065HLBackupLeft;
      FP    #tmpOldAlarm.W065HLBackupLeft;
      JC    LALG;
      L     B#(4, 36);
      A     #tmpNewAlarm.A066HLBackupRight;
      FP    #tmpOldAlarm.A066HLBackupRight;
      JC    LALG;
      L     B#(4, 37);
      A     #tmpNewAlarm.W067HLBackupRight;
      FP    #tmpOldAlarm.W067HLBackupRight;
      JC    LALG;
      L     B#(4, 38);
      A     #tmpNewAlarm.Ax68InletFull;
      FP    #tmpOldAlarm.Ax68InletFull;
      JC    LALG;
      L     B#(4, 39);
      A     #tmpNewAlarm.Ax69DosMax;
      FP    #tmpOldAlarm.Ax69DosMax;
      JC    LALG;
      L     B#(4, 40);
      A     #tmpNewAlarm.A070CANCOM;
      FP    #tmpOldAlarm.A070CANCOM;
      JC    LALG;
      L     B#(4, 41);
      A     #tmpNewAlarm.A071CANMOD;
      FP    #tmpOldAlarm.A071CANMOD;
      JC    LALG;
      L     B#(4, 42);	//[1.2]
      A     #tmpNewAlarm.A072CANDOUT;
      FP    #tmpOldAlarm.A072CANDOUT;
      JC    LALG;
      L     B#(4, 45);
      A     #tmpNewAlarm.W075WarnTemp;
      FP    #tmpOldAlarm.W075WarnTemp;
      JC    LALG;
      L     B#(4, 46);
      A     #tmpNewAlarm.A076HighTemp;
      FP    #tmpOldAlarm.A076HighTemp;
      JC    LALG;
      L     B#(4, 47);
      A     #tmpNewAlarm.A077DigOut;
      FP    #tmpOldAlarm.A077DigOut;
      JC    LALG;
      L     B#(4, 48);
      A     #tmpNewAlarm.A078Service;
      FP    #tmpOldAlarm.A078Service;
      JC    LALG;
      L     B#(4, 49);
      A     #tmpNewAlarm.A110Gap;
      FP    #tmpOldAlarm.A110Gap;
      JC    LALG;
      JU    LAJ8;
//Enter Log message
LALG: A     #Par.ParLogOff;
      JC    LAST;
      T     #tmpLOGvalue;
      L     #tmpIdx;
      +     -1;
      L     50;
      *I;
      L     #tmpLOGvalue;
      +I;
      T     #tmpLOGvalue;
      L     W#16#FF;
      AW;
      T     #OutAlarmNoLog;
      CALL  "GCS7_LogConvert" (
           ObjectNo                 := #Par.ParObjectNo,
           MsgType                  := #Par.ParMsgType,
           ClassMsgTxt              := #tmpLOGvalue,
           OType                    := 1037);	//LOG Message Converter / Entry / Contains Class and TextNo
//============================================================
//Store Old Alarm from stack tmpOldAlarm to current index to stack
LAST: LAR1  P##tmpOldAlarm;
      L     LD [AR1,P#0.0];
      LAR1  #tmpAddrOut_tmpLCAlarm;
      T     DID [AR1,P#0.0];
//Store Data of Index
      AN    #tmpPxAlarmNoValid;
      JC    LAJ8;
      L     1;
      L     #tmpIdx;
      <>I;
      JC    LAI2;
      A     #tmpPxFault;
      =     #Side1.OutLCFault;
      A     #tmpPxWarning;
      =     #Side1.OutLCWarning;
      JU    LAJ8;
LAI2: L     2;
      L     #tmpIdx;
      <>I;
      JC    LAI3;
      A     #tmpPxFault;
      =     #Side2.OutLCFault;
      A     #tmpPxWarning;
      =     #Side2.OutLCWarning;
      JU    LAJ8;
LAI3: L     3;
      L     #tmpIdx;
      <>I;
      JC    LAI4;
      A     #tmpPxFault;
      =     #Side1Divide.OutLCFault;
      A     #tmpPxWarning;
      =     #Side1Divide.OutLCWarning;
      JU    LAJ8;
LAI4: A     #tmpPxFault;
      =     #Side2Divide.OutLCFault;
      A     #tmpPxWarning;
      =     #Side2Divide.OutLCWarning;
      JU    LAJ8;
//---Next Passage-----
LAJ8: L     #tmpIdx;	//Next Index
      +     1;
      JU    LAJ0;
LAJ9: NOP   0;
NETWORK
TITLE = Command to MDDR
      NOP   0;
//==============================
      A     #CmdFaultReset;
      R     #Par.HelpFlags.OutTestNewAlarm;
      A     #tmpSendDone;
      A     #Command.ResetAlarm;
      R     #Command.ResetAlarm;
      S     #Par.HelpFlags.OutTestNewAlarm;
      A     #tmpSendDone;
      A     #CmdFaultReset;
      R     #CmdFaultReset;
      S     #Command.ResetAlarm;
      R     #Side1.OutAlarmNoValid;
      R     #Side2.OutAlarmNoValid;
      R     #Side1Divide.OutAlarmNoValid;
      R     #Side2Divide.OutAlarmNoValid;
//==============================
      A     #Side1.InEnableDosing;
      =     #Command.S1Start;
      A     #Side1.InRestdischarge;
      =     #Command.S1RestDischarge;
//==============================
      A     #Side2.InEnableDosing;
      =     #Command.S2Start;
      A     #Side2.InRestdischarge;
      =     #Command.S2RestDischarge;
//==============================
      A     #Status.NewDataReady;
      =     #Command.AcceptNewDataReady;
//==============================
      SET;
      =     #Command.CommandReady;
//==============================
      A     #Status.NewRcvData;
      =     #Command.AcceptNewRcvData;
//==============================
      AN    #Status.AcceptNewSendData;
      =     #Command.NewSendData;
NETWORK
TITLE = (Profibus) Send Data
      NOP   0;
//------------------------------------------------
//Test Done: Send Dataset 128 Index 1
      L     #DPData.NoSndDataSet;
      L     128;
      <>I;
      JC    s03A;
      L     #DPData.IdxSndDataSet;
      L     1;
      <>I;
      JC    s28B;
      JU    S28B;	//-->Send 128 Index 2
//------------------------------------------------
//Test Done: Send Dataset 128 Index 2
s28B: L     #DPData.IdxSndDataSet;
      L     2;
      <>I;
      JC    S28A;
      JU    S03A;	//-->Send 3 Index 1
//------------------------------------------------
//Test Done: Send Dataset 3 Index 1
s03A: L     #DPData.NoSndDataSet;
      L     3;
      <>I;
      JC    S28A;	//-->Send 128 Index 1
      L     #DPData.IdxSndDataSet;
      L     1;
      <>I;
      JC    s03B;
      AN    #Status.WrongValue;
      A     #Par.HelpFlags.CmdNewValueS1;
      R     #Par.HelpFlags.CmdNewValueS1;
      R     #Side1.CmdNewValue;
      R     #Side1.CmdNewJob;
      JU    S03B;	//-->Send 3 Index 2
//------------------------------------------------
//Test Done: Send Dataset 3 Index 2
s03B: L     #DPData.IdxSndDataSet;
      L     2;
      <>I;
      JC    S28A;
      AN    #Status.WrongValue;
      A     #Par.HelpFlags.CmdNewValueS2;
      R     #Par.HelpFlags.CmdNewValueS2;
      R     #Side2.CmdNewValue;
      R     #Side2.CmdNewJob;
      JU    S28A;	//-->Send 128 Index 1
//==================================================
//Send Dataset 3 Index 1
S03A: L     3;
      T     #DPData.NoSndDataSet;
      L     1;
      T     #DPData.IdxSndDataSet;
      L     0;
      LAR1  P##DPData;
      T     LD [AR1,P#8.0];
      T     LD [AR1,P#12.0];
      T     LD [AR1,P#16.0];
      T     LD [AR1,P#20.0];
//-- Handshake bit
      L     0;
      AN    #PCWrite.Hsk.AckRegisterSide1;
      JC    S3B1;
      L     2#100000000;
S3B1: AN    #PCWrite.Hsk.AckRollChangeDoneSide1;
      JC    S3B2;
      L     2#1000000000;
      +I;
S3B2: AN    #PCWrite.Hsk.Ack600CalibrationSide1;
      JC    S3B3;
      L     2#10000000000;
      +I;
S3B3: T     #DPData.Data.Byte8_9;
//---
      AN    #Side1.OutManual;
      A     #Side1.CmdNewValue;
      O     #Side1.CmdNewJob;
      JCN   send;
      =     #Par.HelpFlags.CmdNewValueS1;
      L     #DPData.Data.Byte8_9;
      L     2#1;
      OW;
      T     #DPData.Data.Byte8_9;
      L     #Side1.In.InGapAdjustment;
      SLW   8;
      T     #DPData.Data.Byte10_11;
      L     #Side1.In.InGapTopLeft;
      T     #DPData.Data.Byte12_13;
      L     #Side1.In.InGapTopRight;
      T     #DPData.Data.Byte14_15;
      L     #Side1.In.InGapBottomLeft;
      T     #DPData.Data.Byte16_17;
      L     #Side1.In.InGapBottomRight;
      T     #DPData.Data.Byte18_19;
      JU    send;
//==================================================
//Send Dataset 3 Index 2
S03B: L     3;
      T     #DPData.NoSndDataSet;
      L     2;
      T     #DPData.IdxSndDataSet;
      L     0;
      LAR1  P##DPData;
      T     LD [AR1,P#8.0];
      T     LD [AR1,P#12.0];
      T     LD [AR1,P#16.0];
      T     LD [AR1,P#20.0];
//-- Handshake bit
      L     0;
      AN    #PCWrite.Hsk.AckRegisterSide2;
      JC    S3C1;
      L     2#100000000;
S3C1: AN    #PCWrite.Hsk.AckRollChangeDoneSide2;
      JC    S3C2;
      L     2#1000000000;
      +I;
S3C2: AN    #PCWrite.Hsk.Ack600CalibrationSide2;
      JC    S3C3;
      L     2#10000000000;
      +I;
S3C3: T     #DPData.Data.Byte8_9;
//---
      AN    #Side2.OutManual;
      A     #Side2.CmdNewValue;
      O     #Side2.CmdNewJob;
      JCN   send;
      =     #Par.HelpFlags.CmdNewValueS2;
      L     #DPData.Data.Byte8_9;
      L     2#1;
      OW;
      T     #DPData.Data.Byte8_9;
      L     #Side2.In.InGapAdjustment;
      SLW   8;
      T     #DPData.Data.Byte10_11;
      L     #Side2.In.InGapTopLeft;
      T     #DPData.Data.Byte12_13;
      L     #Side2.In.InGapTopRight;
      T     #DPData.Data.Byte14_15;
      L     #Side2.In.InGapBottomLeft;
      T     #DPData.Data.Byte16_17;
      L     #Side2.In.InGapBottomRight;
      T     #DPData.Data.Byte18_19;
      JU    send;
//==================================================
//Send Dataset 128 Index 1
S28A: L     128;
      T     #DPData.NoSndDataSet;
      L     1;
      T     #DPData.IdxSndDataSet;
      L     #Side1.In.InRollsUpCurrent;
      T     #DPData.Data.Byte8_9;
      L     #Side1.In.InRollsLowCurrent;
      T     #DPData.Data.Byte10_11;
      L     0;
      LAR1  P##DPData;
      T     LD [AR1,P#12.0];
      T     LD [AR1,P#16.0];
      T     LD [AR1,P#20.0];
      L     0;
      AN    #Side1.In.InRollsUpUsed;
      JC    S28M;
      L     W#16#100;
      +I;
S28M: AN    #Side1.In.InRollsLowUsed;
      JC    S28N;
      L     W#16#200;
      +I;
S28N: T     #DPData.Data.Byte20_21;
      JU    send;
//==================================================
//Send Dataset 128 Index 2
S28B: L     128;
      T     #DPData.NoSndDataSet;
      L     2;
      T     #DPData.IdxSndDataSet;
      L     #Side2.In.InRollsUpCurrent;
      T     #DPData.Data.Byte8_9;
      L     #Side2.In.InRollsLowCurrent;
      T     #DPData.Data.Byte10_11;
      L     0;
      LAR1  P##DPData;
      T     LD [AR1,P#12.0];
      T     LD [AR1,P#16.0];
      T     LD [AR1,P#20.0];
      L     0;
      AN    #Side2.In.InRollsUpUsed;
      JC    S28m;
      L     W#16#100;
      +I;
S28m: AN    #Side2.In.InRollsLowUsed;
      JC    S28n;
      L     W#16#200;
      +I;
S28n: T     #DPData.Data.Byte20_21;
      JU    send;
//======================================================
//Send Dataset to Profibus
send: CALL  "SIEMENS_BLKMOV" (
           SRCBLK                   := #Command,
           RET_VAL                  := #tmpReturn,
           DSTBLK                   := #DPData.StatusCommand);
      L     #DPData.NoSndDataSet;
      T     #Par.OutNoSndDataSet;
      L     #DPData.IdxSndDataSet;
      T     #Par.OutIdxSndDataSet;
      L     #DPData.NoRcvDataSet;
      T     #Par.OutNoRcvDataSet;
      L     #DPData.IdxRcvDataSet;
      T     #Par.OutIdxRcvDataSet;
      A     #InSimulation;
      JC    sSim;
      CALL  "SIEMENS_DPWR_DAT" (
           LADDR                    := #tmpAddr,
           RECORD                   := #DPData,
           RET_VAL                  := #tmpReturn);
      L     #tmpReturn;
      L     0;
      <>I;
      =     #Par.HelpFlags.OutComFaultSend;
      JU    DP_C;
//write to Simulation
sSim: R     #Par.HelpFlags.OutComFaultSend;
      A     "GCS7_Gr_SimDPtoImage";
      L     P#Q 0.0;
      JC    rDB2;
      OPN   "TEST_IOSimuliOutput";
      L     P#DBX 0.0;
rDB2: L     #Par.ParIOByteNo;
      SLD   3;
      +D;
      T     #tmpAddrIO;
      L     #DPData.StatusCommand;
      LAR1  #tmpAddrIO;
      T     D [AR1,P#0.0];
      LAR1  P##DPData;
      L     LD [AR1,P#4.0];
      LAR1  #tmpAddrIO;
      T     D [AR1,P#4.0];
      LAR1  P##DPData;
      L     LD [AR1,P#8.0];
      LAR1  #tmpAddrIO;
      T     D [AR1,P#8.0];
      LAR1  P##DPData;
      L     LD [AR1,P#12.0];
      LAR1  #tmpAddrIO;
      T     D [AR1,P#12.0];
      LAR1  P##DPData;
      L     LD [AR1,P#16.0];
      LAR1  #tmpAddrIO;
      T     D [AR1,P#16.0];
      LAR1  P##DPData;
      L     LD [AR1,P#20.0];
      LAR1  #tmpAddrIO;
      T     D [AR1,P#20.0];
DP_C: NOP   0;
NETWORK
TITLE = Init Flag #tmpAllAlarmNoValide
      A     #Side1.OutAlarmNoValid;
      A     #Side2.OutAlarmNoValid;
      A(;
      A     #Side1Divide.OutAlarmNoValid;
      ON    #Par.ParSide1Divided;
      );
      A(;
      A     #Side2Divide.OutAlarmNoValid;
      ON    #Par.ParSide2Divided;
      );
      =     #tmpAllAlarmNoValide;
NETWORK
TITLE = States Communication
      NOP   0;
//--- tmpFault   
      A     #OutComFault;
      ON    #Status.RemoteControl;
      AN    #tmpLocal;
      =     #tmpFault;
//===================================
//StOK
//===================================
CS2:  AN    #StOk;
      JC    CS4;
//-Transition to StFault
      A     #tmpFault;	//-->StFault
      JC    CxS4;
      JU    CJ9;	//-->StOK
//===================================
//StFault
//===================================
CxS4: R     #StOk;
      S     #StFault;
      S     "GCS7_Gr_InFaultFlag";	//Gr.InFaultFlag
      S     #tmpHornOn;
      R     #OutEdgeComFault;	//reLOG fault
//---Condition for StOk
CS4:  AN    #StFault;
      S     #StOk;	//Init
      JC    CS2;
      A     #tmpAllAlarmNoValide;
      A     #Par.HelpFlags.OutTestNewAlarm;
      AN    #tmpFault;
      O     #InLocal;
      S     #StOk;
      R     #StFault;
      R     #CmdFaultReset;
      JC    CJ9;	//-->StOK
      A     #tmpAllAlarmNoValide;
      A     #Par.HelpFlags.OutTestNewAlarm;
      R     #OutEdgeComFault;	//reLOG fault
CJ9:  NOP   0;
NETWORK
TITLE = States Side 1
      NOP   0;
//--- tmpFault   
      A     #Side1.OutLCFault;
      O     #OutComFault;
      AN    #tmpLocal;
      =     #tmpFault;
//==================================
//StDisengaged
//==================================
P1S0: AN    #Side1.StDisenaged;
      JC    P1S2;
      A     #tmpFault;
      JC    P1X4;	//--> StFault
      AN    #Status.S1Disengaged;
      R     #Side1.StDisenaged;
      S     #Side1.StEngaged;	//--> StEngaged
      JU    P1J9;
//==================================
//StEngaged
//==================================
P1S2: AN    #Side1.StEngaged;
      JC    P1S4;
      A     #tmpFault;
      JC    P1X4;	//--> StFault
      A     #Status.S1Disengaged;
      R     #Side1.StEngaged;
      S     #Side1.StDisenaged;	//--> StDisenaged
      JU    P1J9;
//==================================
//StFault
//==================================
P1X4: S     #Side1.StFault;
      R     #Side1.StEngaged;
      R     #Side1.StDisenaged;
      S     "GCS7_Gr_InFaultFlag";	//Gr.InFaultFlag
      S     #tmpHornOn;
P1S4: AN    #Side1.StFault;
      S     #Side1.StDisenaged;
      JC    P1S0;
      AN    #tmpFault;
      A     #Side1.OutAlarmNoValid;
      A     #Par.HelpFlags.OutTestNewAlarm;
      O     #tmpLocal;
      R     #Side1.StFault;
      S     #Side1.StDisenaged;	//--> StDisenaged
      JC    P1S0;
P1J9: NOP   0;
NETWORK
TITLE = States Side 2
      NOP   0;
//--- tmpFault   
      A     #Side2.OutLCFault;
      O     #OutComFault;
      AN    #tmpLocal;
      =     #tmpFault;
//==================================
//StDisengaged
//==================================
P2S0: AN    #Side2.StDisenaged;
      JC    P2S2;
      A     #tmpFault;
      JC    P2X4;	//--> StFault
      AN    #Status.S2Disengaged;
      R     #Side2.StDisenaged;
      S     #Side2.StEngaged;	//--> StEngaged
      JU    P2J9;
//==================================
//StEngaged
//==================================
P2S2: AN    #Side2.StEngaged;
      JC    P2S4;
      A     #tmpFault;
      JC    P2X4;	//--> StFault
      A     #Status.S2Disengaged;
      R     #Side2.StEngaged;
      S     #Side2.StDisenaged;	//--> StDisenaged
      JU    P2J9;
//==================================
//StFault
//==================================
P2X4: S     #Side2.StFault;
      R     #Side2.StEngaged;
      R     #Side2.StDisenaged;
      S     "GCS7_Gr_InFaultFlag";	//Gr.InFaultFlag
      S     #tmpHornOn;
P2S4: AN    #Side2.StFault;
      S     #Side2.StDisenaged;
      JC    P2S0;
      AN    #tmpFault;
      A     #Side2.OutAlarmNoValid;
      A     #Par.HelpFlags.OutTestNewAlarm;
      O     #tmpLocal;
      R     #Side2.StFault;
      S     #Side2.StDisenaged;	//--> StDisenaged
      JC    P2S0;
P2J9: NOP   0;
NETWORK
TITLE = States Side1Divide
      NOP   0;
//--- tmpFault   
      A     #Side1Divide.OutLCFault;
      O     #OutComFault;
      AN    #tmpLocal;
      =     #tmpFault;
//==================================
//StDisengaged
//==================================
P3S0: AN    #Side1Divide.StDisenaged;
      JC    P3S2;
      A     #tmpFault;
      A     #Par.ParSide1Divided;
      JC    P3X4;	//--> StFault
      AN    #Status.S1Disengaged;
      A     #Par.ParSide1Divided;
      R     #Side1Divide.StDisenaged;
      S     #Side1Divide.StEngaged;	//--> StEngaged
      JU    P3J9;
//==================================
//StEngaged
//==================================
P3S2: AN    #Side1Divide.StEngaged;
      JC    P3S4;
      A     #tmpFault;
      JC    P3X4;	//--> StFault
      A     #Status.S1Disengaged;
      ON    #Par.ParSide1Divided;
      R     #Side1Divide.StEngaged;
      S     #Side1Divide.StDisenaged;	//--> StDisenaged
      JU    P3J9;
//==================================
//StFault
//==================================
P3X4: S     #Side1Divide.StFault;
      R     #Side1Divide.StEngaged;
      R     #Side1Divide.StDisenaged;
      S     "GCS7_Gr_InFaultFlag";	//Gr.InFaultFlag
      S     #tmpHornOn;
P3S4: AN    #Side1Divide.StFault;
      S     #Side1Divide.StDisenaged;
      JC    P3S0;
      AN    #tmpFault;
      A     #Side1Divide.OutAlarmNoValid;
      O     #tmpLocal;
      ON    #Par.ParSide1Divided;
      R     #Side1Divide.StFault;
      S     #Side1Divide.StDisenaged;	//--> StDisenaged
      JC    P3S0;
P3J9: NOP   0;
NETWORK
TITLE = States Side2Divide
      NOP   0;
//--- tmpFault   
      A     #Side2Divide.OutLCFault;
      O     #OutComFault;
      AN    #tmpLocal;
      =     #tmpFault;
//==================================
//StDisengaged
//==================================
P4S0: AN    #Side2Divide.StDisenaged;
      JC    P4S2;
      A     #tmpFault;
      A     #Par.ParSide2Divided;
      JC    P4X4;	//--> StFault
      AN    #Status.S2Disengaged;
      A     #Par.ParSide2Divided;
      R     #Side2Divide.StDisenaged;
      S     #Side2Divide.StEngaged;	//--> StEngaged
      JU    P4J9;
//==================================
//StEngaged
//==================================
P4S2: AN    #Side2Divide.StEngaged;
      JC    P4S4;
      A     #tmpFault;
      JC    P4X4;	//--> StFault
      A     #Status.S2Disengaged;
      ON    #Par.ParSide2Divided;
      R     #Side2Divide.StEngaged;
      S     #Side2Divide.StDisenaged;	//--> StDisenaged
      JU    P4J9;
//==================================
//StFault
//==================================
P4X4: S     #Side2Divide.StFault;
      R     #Side2Divide.StEngaged;
      R     #Side2Divide.StDisenaged;
      S     "GCS7_Gr_InFaultFlag";	//Gr.InFaultFlag
      S     #tmpHornOn;
P4S4: AN    #Side2Divide.StFault;
      S     #Side2Divide.StDisenaged;
      JC    P4S0;
      AN    #tmpFault;
      A     #Side2Divide.OutAlarmNoValid;
      O     #tmpLocal;
      ON    #Par.ParSide2Divided;
      R     #Side2Divide.StFault;
      S     #Side2Divide.StDisenaged;	//--> StDisenaged
      JC    P4S0;
P4J9: NOP   0;
NETWORK
TITLE = Warning/ Horn On
      NOP   0;
//---tmpWarning
      A     #Side1.OutLCWarning;
      AN    #Side1.StFault;
      O;
      A     #Side2.OutLCWarning;
      AN    #Side1.StFault;
      O;
      A     #Side1Divide.OutLCWarning;
      AN    #Side1Divide.StFault;
      O;
      A     #Side2Divide.OutLCWarning;
      AN    #Side2Divide.StFault;
      FP    #OutWarning;
      AN    #tmpLocal;
      S     #tmpHornOn;
//---Horn On-----------------------------
      AN    #tmpHornOn;
      O     #tmpLocal;
      JC    HOJ9;
      CALL  "SYS_Horn_Code" (
           FcCode                   := 1,
           ParObjectType            := 1037,
           ParObjectNo              := #Par.ParObjectNo,
           ParHornCode              := #Par.ParHornCode);
HOJ9: NOP   0;
NETWORK
TITLE = Log2: OutFaultRelevant / Message ComFault / FaultCanceled
//MessageClass Fault Canceled
      A     #Side1.StFault;
      O     #Side2.StFault;
      O     #Side1Divide.StFault;
      O     #Side2Divide.StFault;
      O     #StFault;
      FN    #OutFaultRelevant;
      L     B#(3, 255);	// MessageClass Operate fault cancelled
      JC    LOG;
      A     #StFault;
      FP    #OutEdgeComFault;
      JCN   LOUT;
      L     B#(1, 250);	//Fault Remote Control DP Mode
      AN    #Status.RemoteControl;
      AN    #OutComFault;
      JC    LOG;
      L     B#(1, 251);	//Comunication Fault
LOG:  A     #Par.ParLogOff;	//---Set LOG Message
      JC    LOUT;
      T     #tmpLOGvalue;
      L     W#16#FF;
      AW;
      T     #OutAlarmNoLog;
      CALL  "GCS7_LogConvert" (
           ObjectNo                 := #Par.ParObjectNo,
           MsgType                  := #Par.ParMsgType,
           ClassMsgTxt              := #tmpLOGvalue,
           OType                    := 1037);	//LOG Message Converter / Entry / Contains Class and TextNo
LOUT: NOP   0;
NETWORK
TITLE = State Code Element
      L     43;	//Code: #StOk.DPFault
      A     #OutComFault;
      A     #StOk;
      JC    STC;
      L     3;	//Code: #StOk
      A     #StOk;
      JC    STC;
      L     32;	//Code: fault
STC:  L     #StCode;	//Old state code
      TAK;
      T     #StCode;	//Save state code
      <>I;
      L     3;	//Load code for CBit methode
      CC    "SYS_CBitCtrl";
NETWORK
TITLE = State Code Side 1
      L     44;	//Code: StDisenaged.DPFault
      A     #OutComFault;
      A     #Side1.StEngaged;
      JC    S1C;
      L     14;	//Code: StEnaged.Warning
      A     #Side1.OutLCWarning;
      A     #Side1.StEngaged;
      JC    S1C;
      L     4;	//Code: StEnaged
      A     #Side1.StEngaged;
      JC    S1C;
      L     41;	//Code: StDisenaged.DPFault
      A     #OutComFault;
      A     #Side1.StDisenaged;
      JC    S1C;
      L     11;	//Code: StDisenaged.Warning
      A     #Side1.OutLCWarning;
      A     #Side1.StDisenaged;
      JC    S1C;
      L     1;	//Code: StDisenaged
      A     #Side1.StDisenaged;
      JC    S1C;
      L     32;	//Code: StFault
S1C:  T     #Side1.StCode;	// Save state code
NETWORK
TITLE = State Code Side 2
      L     44;	//Code: StDisenaged.DPFault
      A     #OutComFault;
      A     #Side2.StEngaged;
      JC    S2C;
      L     14;	//Code: StEnaged.Warning
      A     #Side2.OutLCWarning;
      A     #Side2.StEngaged;
      JC    S2C;
      L     4;	//Code: StEnaged
      A     #Side2.StEngaged;
      JC    S2C;
      L     41;	//Code: StDisenaged.DPFault
      A     #OutComFault;
      A     #Side2.StDisenaged;
      JC    S2C;
      L     11;	//Code: StDisenaged.Warning
      A     #Side2.OutLCWarning;
      A     #Side2.StDisenaged;
      JC    S2C;
      L     1;	//Code: StDisenaged
      A     #Side2.StDisenaged;
      JC    S2C;
      L     32;	//Code: StFault
S2C:  T     #Side2.StCode;	// Save state code
NETWORK
TITLE = State Code Side1Divide
      L     44;	//Code: StDisenaged.DPFault
      A     #OutComFault;
      A     #Side1Divide.StEngaged;
      JC    S3C;
      L     14;	//Code: StEnaged.Warning
      A     #Side1Divide.OutLCWarning;
      A     #Side1Divide.StEngaged;
      JC    S3C;
      L     4;	//Code: StEnaged
      A     #Side1Divide.StEngaged;
      JC    S3C;
      L     41;	//Code: StDisenaged.DPFault
      A     #OutComFault;
      A     #Side1Divide.StDisenaged;
      JC    S3C;
      L     11;	//Code: StDisenaged.Warning
      A     #Side1Divide.OutLCWarning;
      A     #Side1Divide.StDisenaged;
      JC    S3C;
      L     1;	//Code: StDisenaged
      A     #Side1Divide.StDisenaged;
      JC    S3C;
      L     32;	//Code: StFault
S3C:  T     #Side1Divide.StCode;	// Save state code
NETWORK
TITLE = State Code Side2Divide
      L     44;	//Code: StDisenaged.DPFault
      A     #OutComFault;
      A     #Side2Divide.StEngaged;
      JC    S4C;
      L     14;	//Code: StEnaged.Warning
      A     #Side2Divide.OutLCWarning;
      A     #Side2Divide.StEngaged;
      JC    S4C;
      L     4;	//Code: StEnaged
      A     #Side2Divide.StEngaged;
      JC    S4C;
      L     41;	//Code: StDisenaged.DPFault
      A     #OutComFault;
      A     #Side2Divide.StDisenaged;
      JC    S4C;
      L     11;	//Code: StDisenaged.Warning
      A     #Side2Divide.OutLCWarning;
      A     #Side2Divide.StDisenaged;
      JC    S4C;
      L     1;	//Code: StDisenaged
      A     #Side2Divide.StDisenaged;
      JC    S4C;
      L     32;	//Code: StFault
S4C:  T     #Side2Divide.StCode;	// Save state code
NETWORK
TITLE = Comunication : Maintanance Counter 
// Maintanance Counter OutCntFault
      A     #StFault;
      FP    #VarEdgeStFault;
      JCN   MCJO;
      L     #OutCntFault;
      +     L#1;
      T     #OutCntFault;
// Maintanance Counter Fault Time
MCJO: ON    #StFault;
      ON    "GCS7_Gr_OutTick1s";	// Increment all s
      JC    MCJ2;
      L     #OutTimeFaulted;
      +     L#1;
      T     #OutTimeFaulted;
MCJ2: NOP   0;
NETWORK
TITLE = Side1: Maintanance Counter 
// Maintanance Counter OutCntFault
      A     #Side1.StFault;
      FP    #Side1.VarEdgeStFault;
      JCN   M1JO;
      L     #Side1.OutCntFault;
      +     L#1;
      T     #Side1.OutCntFault;
// Maintanance Counter Fault Time
M1JO: ON    #Side1.StFault;
      ON    "GCS7_Gr_OutTick1s";	// Increment all s
      JC    M1J2;
      L     #Side1.OutTimeFaulted;
      +     L#1;
      T     #Side1.OutTimeFaulted;
M1J2: NOP   0;
NETWORK
TITLE = Side2: Maintanance Counter 
// Maintanance Counter OutCntFault
      A     #Side2.StFault;
      FP    #Side2.VarEdgeStFault;
      JCN   M2JO;
      L     #Side2.OutCntFault;
      +     L#1;
      T     #Side2.OutCntFault;
// Maintanance Counter Fault Time
M2JO: ON    #Side2.StFault;
      ON    "GCS7_Gr_OutTick1s";	// Increment all s
      JC    M2J2;
      L     #Side2.OutTimeFaulted;
      +     L#1;
      T     #Side2.OutTimeFaulted;
M2J2: NOP   0;
NETWORK
TITLE = Side1Divide Maintanance Counter 
// Maintanance Counter OutCntFault
      A     #Side1Divide.StFault;
      FP    #Side1Divide.VarEdgeStFault;
      JCN   M3JO;
      L     #Side1Divide.OutCntFault;
      +     L#1;
      T     #Side1Divide.OutCntFault;
// Maintanance Counter Fault Time
M3JO: ON    #Side1Divide.StFault;
      ON    "GCS7_Gr_OutTick1s";	// Increment all s
      JC    M3J2;
      L     #Side1Divide.OutTimeFaulted;
      +     L#1;
      T     #Side1Divide.OutTimeFaulted;
M3J2: NOP   0;
NETWORK
TITLE = Side2Divide Maintanance Counter 
// Maintanance Counter OutCntFault
      A     #Side2Divide.StFault;
      FP    #Side2Divide.VarEdgeStFault;
      JCN   M4JO;
      L     #Side2Divide.OutCntFault;
      +     L#1;
      T     #Side2Divide.OutCntFault;
// Maintanance Counter Fault Time
M4JO: ON    #Side2Divide.StFault;
      ON    "GCS7_Gr_OutTick1s";	// Increment all s
      JC    M4J2;
      L     #Side2Divide.OutTimeFaulted;
      +     L#1;
      T     #Side2Divide.OutTimeFaulted;
M4J2: NOP   0;
NETWORK
TITLE = Global End 
      NOP   0;
//Clear Flag
      A     #tmpAllAlarmNoValide;
      R     #Par.HelpFlags.OutTestNewAlarm;
//--Output for group 
      AN    #InLocal;
      A     #OutComFault;
      S     "GCS7_Gr_InDPFault";
      NOP   0;
END_FUNCTION_BLOCK

